						FB_Move.BCGapMove:=TRUE;
						FB_Move();
						HysteresisMoving:=TRUE;		
						n_state:=1;	
					END_IF
				1:
					btn_UserGapMove:=FALSE;
					FB_Move();
					IF NOT FB_Move.BCGapDone THEN			(*还未运动到位置,运动过程中*)
						Led_Run:=TRUE;
						n_state:=1;
					ELSE									
						n_state:=2;							(*转到下一步，运动到最终位置*)
						FB_Move.BCGapMove:=FALSE;
						//Led_Run:=FALSE;
					END_IF
				2:
					FB_Move.BCGapReset:=FALSE;
					FB_Move.Mode:=5;						//1.gap;2.single;3.taper;4.debug;5.BCGap&UserMode
					FB_Move.CoupleState:=st_Couple;			
					FB_Move.PowerState:=st_Power;			
					FB_Move.BCGapMove:=TRUE;
					//直接走到目标位置，已经走到位置的，可以继续下命令，只不过它不在走了而已
					FB_Move.BCLeftTopPosition:=LeftTopLinPositionNewTemp;	
					FB_Move.BCRightTopPosition:=RightTopLinPositionNewTemp;
					FB_Move.BCLeftBottomPosition:=LeftBottomLinPositionNewTemp;
					FB_Move.BCRightBottomPosition:=RightBottomLinPositionNewTemp;
					//
					//目标速度赋值
					IF NormalGapMode THEN
						FB_Move.BCLeftTopVelocity:=UserGapVelocityNew/2;
						FB_Move.BCRightTopVelocity:=UserGapVelocityNew/2;
						FB_Move.BCLeftBottomVelocity:=UserGapVelocityNew/2;
						FB_Move.BCRightBottomVelocity:=UserGapVelocityNew/2;
					ELSIF IDTaperMode THEN
						FB_Move.BCLeftTopVelocity:=UserTaperVelocityNew/2;
						FB_Move.BCRightTopVelocity:=UserTaperVelocityNew/2;
						FB_Move.BCLeftBottomVelocity:=UserTaperVelocityNew/2;
						FB_Move.BCRightBottomVelocity:=UserTaperVelocityNew/2;
					ELSIF BLTaperMode THEN
						FB_Move.BCLeftTopVelocity:=BLUserTaperVelocityNew*IDTaperAndBLTaperScale/4;
						FB_Move.BCRightTopVelocity:=BLUserTaperVelocityNew*IDTaperAndBLTaperScale/4;
						FB_Move.BCLeftBottomVelocity:=BLUserTaperVelocityNew*IDTaperAndBLTaperScale/4;
						FB_Move.BCRightBottomVelocity:=BLUserTaperVelocityNew*IDTaperAndBLTaperScale/4;
					ELSE
						FB_Move.BCLeftTopVelocity:=0;
						FB_Move.BCRightTopVelocity:=0;
						FB_Move.BCLeftBottomVelocity:=0;
						FB_Move.BCRightBottomVelocity:=0;
					END_IF
					FB_Move();							
					n_state:=3;
				3:
					FB_Move();
					IF NOT FB_Move.BCGapDone THEN			(*还未运动到位置,运动过程中*)
						Led_Run:=TRUE;
						n_state:=3;
					ELSE									
						n_state:=88;							(*运动到了最终位置*)
					END_IF
					(*
					IF NOT Unreach_LS_Bottom THEN
						n_state:=88;							(*在运动过程中如果碰到下限位，则也转到下一步，运动到最终位置*)
						FB_Move.BCGapMove_2:=FALSE;
					END_IF
					*)
				88:
					btn_UserGapMove:=FALSE;					
					Led_Run:=FALSE;
					n_state:=0;
					HysteresisMoving:=FALSE;
			END_CASE
		END_IF
	//
	//FB_Move.BCLeftTopPosition等四轴位置监控
	//
END_IF

IF btn_UserGapStop OR btn_Reset THEN
	FB_Move.BCGapReset:=TRUE;
	FB_Move();	
	btn_UserGapMove:=FALSE;	
	m_state:=0;	
	n_state:=0;	
	HysteresisMoving:=FALSE;
	CASE s_state OF
			0:
				FB_Stop.Mode:=5;	
				FB_Stop.CoupleState:=st_Couple;	
				FB_Stop.PowerState:=st_Power;
				FB_Stop.BCGapStop:=TRUE;
				FB_Stop();	
				s_state:=1;
			1:
				FB_Stop();
				IF NOT FB_Stop.BCGapDone THEN
					s_state:=1;
				ELSE
					s_state:=88;
				END_IF
			88:
				btn_UserGapStop:=FALSE;	
				FB_Move.BCGapReset:=FALSE;
				btn_reset:=FALSE;
				s_state:=0;
		END_CASE
END_IF

(*触发限位开关后，相当于点击了Stop按钮*)
FTrig_ReachLS(CLK:=Unreach_LS_Far AND Unreach_LS_Near);
IF FTrig_ReachLS.Q THEN
	btn_UserGapStop:=TRUE;
END_IF
END_ACTION

ACTION A_SpectroscopyScanningMotion:
(*输入保护*)
IF SS_Move AND SSMotionMode AND NOT RegularMotionMode THEN
	IF NOT inRange_SS_StepSize THEN
		SS_Stop:=TRUE;
		SS_Move:=FALSE;
		Error:=TRUE;
		ErrorId:=805;
		ErrorDescription:='target StepSize out of range,please check';
		RETURN;
	ELSE
		//SS_Stop:=FALSE;
		Error:=FALSE;
		ErrorId:=0;
		ErrorDescription:='';	
	END_IF
	//
	IF NOT inRange_SS_StepNumber THEN
		SS_Stop:=TRUE;
		SS_Move:=FALSE;
		Error:=TRUE;
		ErrorId:=806;
		ErrorDescription:='target StepNumber out of range,please check';
		RETURN;
	ELSE
		//SS_Stop:=FALSE;
		Error:=FALSE;
		ErrorId:=0;
		ErrorDescription:='';	
	END_IF
	IF NOT inRange_SS_StepVelocity THEN
		SS_Stop:=TRUE;
		SS_Move:=FALSE;
		Error:=TRUE;
		ErrorId:=807;
		ErrorDescription:='target StepVelocity out of range,please check';
		RETURN;
	ELSE
		//SS_Stop:=FALSE;
		Error:=FALSE;
		ErrorId:=0;
		ErrorDescription:='';	
	END_IF
	IF NOT inRange_StepEachTime_ms THEN
		SS_Stop:=TRUE;
		SS_Move:=FALSE;
		Error:=TRUE;
		ErrorId:=808;
		ErrorDescription:='target StepEachTime_ms out of range,please check';
		RETURN;
	ELSE
		//SS_Stop:=FALSE;
		Error:=FALSE;
		ErrorId:=0;
		ErrorDescription:='';	
	END_IF
END_IF
(*单步时长转换*)
StepEachTime:=INT_TO_TIME(StepEachTime_ms);
SS_TON(PT:=StepEachTime);
(*上升沿触发，初始SS位置=当前磁间隙*)
RTRG_SS_StartPositionDisplay(CLK:=SS_Move);
IF RTRG_SS_StartPositionDisplay.Q THEN
	SS_StartPositionDisplay:=UserGapPositionDisplay;
	SS_InitStartPositionDone:=TRUE;
END_IF
(*SS主程序*)
IF InitPowerDone AND InitCompensationDatasDone AND SS_Move AND SS_InitStartPositionDone THEN
	IF NOT st_Power THEN
		ErrorID:=1501;
		Error:=TRUE;
		ErrorDescription:='Plz PowerOn Frist';
		LED_Error:=TRUE;
		//btn_UserGapMove:=FALSE;
		RETURN;
	ELSE
		ErrorID:=0;
		Error:=FALSE;
		ErrorDescription:='';
		LED_Error:=FALSE;
		//btn_UserGapMove:=TRUE;
	END_IF	
CASE SS_MoveState OF
		0:
				//UserGapPositionNew:=UserGapPositionDisplay+SS_StepSize;
				UserGapPositionNew:=SS_StartPositionDisplay+SS_StepSize*(SS_currentStep+1);
				A_InitCompensationData();
				FB_Move.Mode:=5;						//1.gap;2.single;3.taper;4.debug;5.BCGap&UserMode
				FB_Move.CoupleState:=st_Couple;			
				FB_Move.PowerState:=st_Power;							
				FB_Move.BCLeftTopPosition:=LeftTopLinPositionNew;
				FB_Move.BCLeftTopVelocity:=SS_StepVelocity/2;
				FB_Move.BCRightTopPosition:=RightTopLinPositionNew;
				FB_Move.BCRightTopVelocity:=SS_StepVelocity/2;
				FB_Move.BCLeftBottomPosition:=LeftBottomLinPositionNew;
				FB_Move.BCLeftBottomVelocity:=SS_StepVelocity/2;
				FB_Move.BCRightBottomPosition:=RightBottomLinPositionNew;
				FB_Move.BCRightBottomVelocity:=SS_StepVelocity/2;		
				FB_Move.BCGapMove:=TRUE;
				FB_Move();
				SS_MoveState:=1;
		1:
				SS_TON.IN:=TRUE;
				FB_Move();
				IF FB_Move.GapMoving AND NOT SS_TimeCountBegin THEN
					SS_StepSystemTime_Begin[SS_currentStep]:=F_GetSysTime();
					SS_TimeCountBegin:=TRUE;
				END_IF
				IF NOT FB_Move.BCGapDone THEN			
					Led_Run:=TRUE;
					SS_MoveState:=1;
				ELSE									
					SS_MoveState:=66;
					SS_StepSystemTime_End[SS_currentStep]:=F_GetSysTime();
					SS_StepCountTime[SS_currentStep]:=SS_StepSystemTime_End[SS_currentStep]-SS_StepSystemTime_Begin[SS_currentStep];
					SS_TimeCountBegin:=FALSE;
				END_IF
		66:
				SS_currentStep:=SS_currentStep+1;			
				Led_Run:=FALSE;
				IF SS_currentStep=SS_StepNumber THEN								
					SS_MoveState:=88;
				END_IF
				IF SS_currentStep<SS_StepNumber THEN
					SS_MoveState:=77;
				END_IF
		77://等待单步时长够
				IF SS_TON.Q THEN
					SS_TON.IN:=FALSE;
					SS_MoveState:=0;
				END_IF
		88:
				SS_TON.IN:=FALSE;
				SS_Move:=FALSE;	
				Led_Run:=FALSE;
				SS_MoveState:=0;
				SS_currentStep:=0;
				SS_InitStartPositionDone:=FALSE;
				//SS_StepSystemTime[SS_StepNumber]:=F_GetSysTime();
	END_CASE
END_IF
(*获取每一步耗时*)
//FOR	m:= 0 TO SS_StepNumber DO
//	SS_StepCountTime[m]:=(SS_StepSystemTime_End[m]-SS_StepSystemTime_Begin[m]);
//END_FOR

(*STOP*)
IF SS_Stop OR btn_reset THEN
	FB_Move.BCGapReset:=TRUE;
	FB_Move();	
	SS_Move:=FALSE;	
	SS_MoveState:=0;	
	CASE SS_StopState OF
			0:
				FB_Stop.Mode:=5;						
				FB_Stop.CoupleState:=st_Couple;		
				FB_Stop.PowerState:=st_Power;			
				FB_Stop.BCGapStop:=TRUE;			
				FB_Stop();						
				SS_StopState:=1;
			1:
				FB_Stop();
				IF NOT FB_Stop.BCGapDone THEN		
					SS_StopState:=1;
				ELSE							
					SS_StopState:=88;
				END_IF
			88:
				SS_Stop:=FALSE;					
				FB_Move.BCGapReset:=FALSE;		
				SS_StopState:=0;
				btn_reset:=FALSE;
				//SS_Stop2:=FALSE;
		END_CASE
END_IF

(*触发限位开关后，相当于点击了Stop按钮*)
FTrig_ReachLS(CLK:=Unreach_LS_Far AND Unreach_LS_Near);
IF FTrig_ReachLS.Q THEN
	SS_Stop:=TRUE;
END_IF
END_ACTION

ACTION A_TaperMotionProtection:
(*如果该ID没有taper需求，则TaperFunctionSolidOn=FALSE，则判定taperOrNot和BLTaperOrNot都为FALSE*)
IF NOT TaperFunctionSolidOn THEN
	TaperOrNot:=FALSE;
	BLTaperOrNot:=FALSE;
END_IF
(*若GAP将有变化，首先检测TAPER是否超出阈值，若超出，则报错，提示必须先将TAPER回归到0，才可以改变GAP*)
IF NormalGapMode OR IDTaperMode THEN 
	IF NOT (Global_ChainProtection_MPS_Triggered OR Global_ChainProtection_EPS_Triggered) THEN//在触发联锁保护后，taper保护关闭
		IF ABS(UserGapPositionNew-UserGapPositionDisplay)>Threshold_GapChangeFlag AND btn_UserGapMove THEN
			IF UserTaperPositionDisplay>Threshold_TaperChangeFlag THEN
				btn_UserGapStop:=TRUE;
				btn_UserGapMove:=FALSE;
				Error:=TRUE;
				ErrorId:=809;
				ErrorDescription:='Please Move Taper to zero first before move gap';
				RETURN;
			END_IF
		END_IF
	END_IF
END_IF
IF BLTaperMode THEN
		IF NOT (Global_ChainProtection_MPS_Triggered OR Global_ChainProtection_EPS_Triggered) THEN//在触发联锁保护后，taper保护关闭
		IF ABS(UserGapPositionNew-UserGapPositionDisplay)>Threshold_GapChangeFlag AND btn_UserGapMove THEN
			IF BLUserTaperPositionDisplay>Threshold_TaperChangeFlag THEN
				btn_UserGapStop:=TRUE;
				btn_UserGapMove:=FALSE;
				Error:=TRUE;
				ErrorId:=810;
				ErrorDescription:='Please Move Taper to zero first before move gap';
				RETURN;
			END_IF
		END_IF
	END_IF
END_IF
(*若GAP将有变化,检测taper功能开关有没有关，要是没有关，提示先关闭*)
IF NOT (Global_ChainProtection_MPS_Triggered OR Global_ChainProtection_EPS_Triggered) THEN//在触发联锁保护后，taper保护关闭
	IF ABS(UserGapPositionNew-UserGapPositionDisplay)>Threshold_GapChangeFlag AND btn_UserGapMove THEN
		IF TaperOrNot OR BLTaperOrNot THEN
			btn_UserGapStop:=TRUE;
			btn_UserGapMove:=FALSE;
			Error:=TRUE;
			ErrorId:=811;
			ErrorDescription:='Please turn off taper function before move gap';
			RETURN;
		END_IF
	END_IF
END_IF
(*Taper和gap连锁限制性保护。比如11mm时候如果taper，入口端gap变小，会有压真空盒的问题。设置保护；在大间隙同样保护*)
IF IDTaperMode THEN
	IF NOT (Global_ChainProtection_MPS_Triggered OR Global_ChainProtection_EPS_Triggered)  THEN//在触发联锁保护后，taper保护关闭
		IF UserGapPositionNew-TaperAndGapSafetyfactor*TaperAndGapSafetyScale*UserTaperPositionNew<(min_UserGapPositionNew+TaperAndGapSafetyMinGapMargin)
			OR UserGapPositionNew+TaperAndGapSafetyfactor*TaperAndGapSafetyScale*UserTaperPositionNew>(max_UserGapPositionNew-TaperAndGapSafetyMinGapMargin) THEN
				 IF btn_UserGapMove THEN
					btn_UserGapStop:=TRUE;
					btn_UserGapMove:=FALSE;
					Error:=TRUE;
					ErrorId:=812;
					ErrorDescription:='Target taper is too big at current Gap';
					RETURN;
				END_IF
		END_IF
	END_IF
END_IF
IF BLTaperMode THEN
	IF NOT (Global_ChainProtection_MPS_Triggered OR Global_ChainProtection_EPS_Triggered)  THEN//在触发联锁保护后，taper保护关闭
		IF UserGapPositionNew-BLUserTaperPositionNew/2<(min_UserGapPositionNew+TaperAndGapSafetyMinGapMargin)
			OR UserGapPositionNew+BLUserTaperPositionNew/2>(max_UserGapPositionNew-TaperAndGapSafetyMinGapMargin) THEN
				 IF btn_UserGapMove THEN
					btn_UserGapStop:=TRUE;
					btn_UserGapMove:=FALSE;
					Error:=TRUE;
					ErrorId:=813;
					ErrorDescription:='Target taper is too big at current Gap';
					RETURN;
				END_IF
		END_IF
	END_IF
END_IF
(*Taper和gap连锁限制性保护。大间隙taper过大，有触碰真空盒问题，保护*)
END_ACTION

ACTION A_TaperParametersInit:
// 先做模式判断
NormalGapMode := NOT TaperOrNot AND NOT BLTaperOrNot;
IDTaperMode := TaperOrNot AND NOT BLTaperOrNot;
BLTaperMode := NOT TaperOrNot AND BLTaperOrNot;
//TaperOrNot和BLTaperOrNot互斥，只能选择其中一个
trig_TaperOrNot(CLK := TaperOrNot);
trig_BLTaperOrNot(CLK := BLTaperOrNot);
IF trig_TaperOrNot.Q THEN
    BLTaperOrNot := FALSE;
ELSIF trig_BLTaperOrNot.Q THEN
    TaperOrNot := FALSE;
END_IF;

//插入件taper/线站taper
IDTaperAndBLTaperScale:=L_Center2Motor/L_HalfGirder;
//插入件taper模式下，入口被动减小的距离，也即a
TaperAndGapSafetyScale:=DINT_TO_LREAL(LREAL_TO_DINT(((L_HalfGirder-L_Center2Motor)/(2*L_Center2Motor))*100000))/100000;

//线站模式下，最大taper由参数表决定，ID模式的最大tape由scale计算得到
max_UserTaperPositionNew:=DINT_TO_LREAL(LREAL_TO_DINT((max_BLUserTaperPositionNew*IDTaperAndBLTaperScale)*100000))/100000;
max_UserTaperVelocityNew:=DINT_TO_LREAL(LREAL_TO_DINT((max_BLUserTaperVelocityNew)*100000))/100000;
//最小taper固定位0
min_UserTaperPositionNew:=0;
min_UserTaperVelocityNew:=0;
END_ACTION

END_PROGRAM

// ---- POUs/MAIN.TcPOU
PROGRAM MAIN
VAR
	pbGapMode: BOOL:=FALSE;
	pbTaperMode: BOOL:=FALSE;
	pbSingleCarrierMode: BOOL:=FALSE;
	pbDebugMode:BOOL:=FALSE;
	pbBCGapMode:BOOL:=FALSE;
	fb_led_Show: FB_LedShow;
	CPMU_PLC_Reset: PLC_Reset;
	d_state: DINT;
	CPMU_PLC_Start: PLC_Start;
	powerStatus:BOOL;

(*TwinSAFE*)
	Safe_run AT%Q*:BOOL;
	Err_Ack AT %Q*:BOOL;
	Estop_RunAndRestart AT %Q*:BOOL;
	AX5805_Error_Ack AT %Q*:BOOL;
	Led_Run  AT %Q*:BOOL;
	Led_Error  AT %Q*:BOOL;

	FB_ERROR AT%I*:BOOL;
	COM_ERROR AT%I*:BOOL;
	//OUT_ERROR AT%I*:BOOL;
	Estop_Out AT%I*:BOOL;

	SafeStatus:INT;
	SafePLCRunOK: BOOL;
	fb_ton: TON;
	fb_ton2: TON;
	fb_ton3: TON;
	fb_ton1: TON;
	fb_ton0: TON;
(*IO*)
	el1808_D1  AT%I* :ARRAY[1..8] OF BOOL;
	el1008 AT%I*:BOOL;
	EStopTrig:BOOL;
(*setAxisPosition*)
	SetAxisPosState: INT;
	FB_Set_AxisPosition:FB_SetAxisPosition;
	fb_ton4: TON;
	fb_ton5: TON;
	fb_ton6: TON;
	SerAxisPositionDone: BOOL;

	i: INT;
	j: INT;

(****RS232***)
	//fbEL6001	: FB_SerialCom;
	moveDoneLeftTop: BOOL;
	moveDoneRightTop: BOOL;
	moveDoneLeftBottom: BOOL;
	moveDoneRightBottom: BOOL;
	moveDoneAllAxis: BOOL;
(**)
	btn_setAxisPosition: BOOL;
	ValueSet_LeftTop:LREAL;
	ValueSet_RightTop:LREAL;
	ValueSet_LeftBottom:LREAL;
	ValueSet_RightBottom:LREAL;
(**)
	RestartTC: TC_Restart;
	
(*recipe*)
	RecipeINT:INT;
	RecipeBOOL:BOOL;
	RecipeManCommands: RecipeManCommands;
	SaveParameter : BOOL;  //保存文件
	LoadParameter : BOOL;  //读取文件
	Save_R_TRIG   : R_TRIG;
	Read_R_TRIG   : R_TRIG;
	loadparameterStatus: INT;
	RecipeBOOL2:BOOL;
	ReturnDwordLoad: DWORD;
	InsertionDeviceName:STRING;
(*UserMode*)
	pbUserMode: BOOL:=TRUE;
	EL1904 AT%I* :ARRAY[1..24] OF BOOL;
	setAxisPositionEnable: BOOL;
	state_loadParameters: INT;
	state_setLEPosBias: INT;
	//
	PositionBiasSet:BOOL;
	MC_SetLEPosBias_LeftTop:MC_WriteParameter;
	MC_SetLEPosBias_RightTop:MC_WriteParameter;
	MC_SetLEPosBias_LeftBottom:MC_WriteParameter;
	MC_SetLEPosBias_RightBottom:MC_WriteParameter;
	PositionBias_LeftTopLin: LREAL:=10.1;
	PositionBias_RightTopLin: LREAL:=10.2;
	PositionBias_LeftBottomLin: LREAL:=10.3;
	PositionBias_RightBottomLin: LREAL:=10.4;
	PositionBias_LeftTop: LREAL:=10.1;
	PositionBias_RightTop: LREAL:=10.2;
	PositionBias_LeftBottom: LREAL:=10.3;
	PositionBias_RightBottom: LREAL:=10.4;

	LoadLEPB_R_TRIG: R_TRIG;
	PositionBiasTON: TON;
	
	//
	OPC_TEST_Bi:BOOL:=TRUE; (*~ (OPC:1:available for OPC Clients) *)
	OPC_TEST_Bi2:BOOL;(*~ (OPC:1:available for OPC Clients) *)
	//
	HasTemperatureSensorOrNot:BOOL;//Only IVU or CPMU
	(*Sensor Reading*)
	TempSensorHardware:DINT:=1;//1:profibus;2:EL3202
	EL3202_Reading AT %I*:ARRAY[0..7] OF INT;	
	EL3202_hReading AT %I*:ARRAY[0..7] OF INT;
	Sensor_Reading_1 AT %I*:ARRAY[0..3] OF BYTE;
	Sensor_Reading_2 AT %I*:ARRAY[0..3] OF BYTE;
	Sensor_Reading_3 AT %I*:ARRAY[0..3] OF BYTE;
	Sensor_Reading_4 AT %I*:ARRAY[0..3] OF BYTE;
	Sensor_Reading_5 AT %I*:ARRAY[0..3] OF BYTE;
	Sensor_Reading_6 AT %I*:ARRAY[0..3] OF BYTE;
	Sensor_Reading_7 AT %I*:ARRAY[0..3] OF BYTE;
	Sensor_Reading_8 AT %I*:ARRAY[0..3] OF BYTE;
	Sensor_Reading_DpState AT %I*:USINT;
	Sensor_Reading_ExtDiagFlag AT %I*:BOOL;
	TemperatureSensors_1:LREAL;
	TemperatureSensors_2:LREAL;
	TemperatureSensors_3:LREAL;
	TemperatureSensors_4:LREAL;
	TemperatureSensors_5:LREAL;
	TemperatureSensors_6:LREAL;
	TemperatureSensors_7:LREAL;
	TemperatureSensors_8:LREAL;
	dut_sensor_datas_1:DUT_SENSOR_DATAS_1;
	dut_sensor_datas_2:DUT_SENSOR_DATAS_2;
	dut_sensor_datas_3:DUT_SENSOR_DATAS_3;
	dut_sensor_datas_4:DUT_SENSOR_DATAS_4;
	dut_sensor_datas_5:DUT_SENSOR_DATAS_5;
	dut_sensor_datas_6:DUT_SENSOR_DATAS_6;
	dut_sensor_datas_7:DUT_SENSOR_DATAS_7;
	dut_sensor_datas_8:DUT_SENSOR_DATAS_8;
	//
	temperature_gradient_2_To_1:LREAL;
	temperature_gradient_3_To_2:LREAL;
	temperature_gradient_5_To_4:LREAL;
	temperature_gradient_6_To_5:LREAL;
	temperature_gradient_max:LREAL;
	//
	temperature_average:LREAL;
	A_SetLinearEncoderPositionBias_Enable: BOOL;
	
	//
	//(*Sensor Reading high temperature*)
	//
	Sensor_Reading_h1 AT %I*:ARRAY[0..3] OF BYTE;
	Sensor_Reading_h2 AT %I*:ARRAY[0..3] OF BYTE;
	Sensor_Reading_h3 AT %I*:ARRAY[0..3] OF BYTE;
	Sensor_Reading_h4 AT %I*:ARRAY[0..3] OF BYTE;
	Sensor_Reading_h5 AT %I*:ARRAY[0..3] OF BYTE;
	Sensor_Reading_h6 AT %I*:ARRAY[0..3] OF BYTE;
	Sensor_Reading_h7 AT %I*:ARRAY[0..3] OF BYTE;
	Sensor_Reading_h8 AT %I*:ARRAY[0..3] OF BYTE;
	Sensor_Reading_DpStateh AT %I*:USINT;
	Sensor_Reading_ExtDiagFlagh AT %I*:BOOL;
	TemperatureSensors_h1:LREAL;
	TemperatureSensors_h2:LREAL;
	TemperatureSensors_h3:LREAL;
	TemperatureSensors_h4:LREAL;
	TemperatureSensors_h5:LREAL;
	TemperatureSensors_h6:LREAL;
	TemperatureSensors_h7:LREAL;
	TemperatureSensors_h8:LREAL;
	dut_sensor_datas_h1:DUT_SENSOR_DATAS_h1;
	dut_sensor_datas_h2:DUT_SENSOR_DATAS_h2;
	dut_sensor_datas_h3:DUT_SENSOR_DATAS_h3;
	dut_sensor_datas_h4:DUT_SENSOR_DATAS_h4;
	dut_sensor_datas_h5:DUT_SENSOR_DATAS_h5;
	dut_sensor_datas_h6:DUT_SENSOR_DATAS_h6;
	dut_sensor_datas_h7:DUT_SENSOR_DATAS_h7;
	dut_sensor_datas_h8:DUT_SENSOR_DATAS_h8;
	//
	temperature_gradient_h2_To_h1:LREAL;
	temperature_gradient_h3_To_h2:LREAL;
	temperature_gradient_h5_To_h4:LREAL;
	temperature_gradient_h6_To_h5:LREAL;
	temperature_gradient_maxh:LREAL;
	//
	temperature_averageh:LREAL;
		//
	temperatureStatus:INT;//0：有传感器度数错误；1:常温；2:低温；3:常温和低温中间态
	CryogenicTemperatureThreshold:LREAL:=82;//82K以下归划分为低温
	RoomTemperatureThreshold:LREAL:=293;//293K以上划分为常温.20摄氏度
	InCryogenicOrNot:BOOL;
	//CPMU cryogenix ON/FF
	CryogenicCompensationOn:BOOL;
	CryogenicCompensationConditionsReady:BOOL;
	CryogenicCompensation_LeftTop:LREAL;
	CryogenicCompensation_RightTop:LREAL;
	CryogenicCompensation_LeftBottom:LREAL;
	CryogenicCompensation_RightBottom:LREAL;
	CryogenicCompensationDone: BOOL;
	
	(**)
	bDriveDiagMessageAndNumber  : BOOL;
	m_GetDriveStatusState:INT;
	GetDriveStatusStateDone:BOOL;
	GetDriveStatusStateError:BOOL;
	GetDriveStatusTON: TON;
	//	
	fb_SoEReadDiagMessage_LeftTop: FB_SoEReadDiagMessage;
	fb_SoEReadDiagMessage_RightTop: FB_SoEReadDiagMessage;
	fb_SoEReadDiagMessage_LeftBottom: FB_SoEReadDiagMessage;
	fb_SoEReadDiagMessage_RightBottom: FB_SoEReadDiagMessage;
	DriveDiagMessage_LeftTop:STRING;
	DriveDiagMessage_RightTop:STRING;
	DriveDiagMessage_LeftBottom:STRING;
	DriveDiagMessage_RightBottom:STRING;
	//
	FB_SoEReadDiagNumber_LeftTop: FB_SoEReadDiagNumber;
	FB_SoEReadDiagNumber_RightTop: FB_SoEReadDiagNumber;
	FB_SoEReadDiagNumber_LeftBottom: FB_SoEReadDiagNumber;
	FB_SoEReadDiagNumber_RightBottom: FB_SoEReadDiagNumber;
	DriveDiagNumber_LeftTop:UDINT;
	DriveDiagNumber_RightTop:UDINT;
	DriveDiagNumber_LeftBottom:UDINT;
	DriveDiagNumber_RightBottom:UDINT;
	bReloadDriveDiagMessageAndNumber: BOOL;
	
	(*load IOC*)
	bExe_load_Prog: BOOL;
	NT_StartProcess_Load: NT_StartProcess;
	Exe_load_step: UINT;
	R_TRIG_ExeLoad: R_TRIG;
	Exe_Load_Done:BOOL;
	(*kill IOC*)
	bExe_Kill_Prog: BOOL;
	NT_StartProcess_Kill: NT_StartProcess;
	Exe_kill_step: UINT;
	R_TRIG_Exekill: R_TRIG;
	Exe_Kill_Done:BOOL;
	LoadOpcIocTON:TON;
	
	LeftTop_2:AXIS_REF;
	RightTop_2:AXIS_REF;
	LeftBottom_2:AXIS_REF;
	RightBottom_2:AXIS_REF;
	Pos_LeftTop_2:LREAL;
	Velo_LeftTop_2:LREAL;
	Pos_RightTop_2:LREAL;
	Velo_RightTop_2:LREAL;
	Pos_LeftBottom_2:LREAL;
	Velo_LeftBottom_2:LREAL;
	Pos_RightBottom_2:LREAL;
	Velo_RightBottom_2:LREAL;
	PosDifference_LeftTop2to1:LREAL;
	PosDifference_RightTop2to1:LREAL;
	PosDifference_LeftBottom2to1:LREAL;
	PosDifference_RightBottom2to1:LREAL;
	//
	//more parameters get:gear;feedback2 direction 
	//
	//GetMoreDriveStatus_FunctionON:BOOL:=TRUE;
	GetDriveStatusTON2: TON;
	//GearNumerator,st182
	st_p182_LeftTop:ST_P182;
	FB_SoERead_GearNumerator_LeftTop: FB_SoERead;
	st_p182_RightTop:ST_P182;
	FB_SoERead_GearNumerator_RightTop: FB_SoERead;
	st_p182_LeftBottom:ST_P182;
	FB_SoERead_GearNumerator_LeftBottom: FB_SoERead;
	st_p182_RightBottom:ST_P182;
	FB_SoERead_GearNumerator_RightBottom: FB_SoERead;
	GearNumeratorGet_LeftTop:UDINT;
	GearNumeratorGet_RightTop:UDINT;
	GearNumeratorGet_LeftBottom:UDINT;
	GearNumeratorGet_RightBottom:UDINT;
	GearNumeratorConfigured_LeftTop:UDINT;
	GearNumeratorConfigured_RightTop:UDINT;
	GearNumeratorConfigured_LeftBottom:UDINT;
	GearNumeratorConfigured_RightBottom:UDINT;
	//GearDenominator,st183
	st_p183_LeftTop:ST_P183;
	FB_SoERead_GearDenominator_LeftTop: FB_SoERead;
	st_p183_RightTop:ST_P183;
	FB_SoERead_GearDenominator_RightTop: FB_SoERead;
	st_p183_LeftBottom:ST_P183;
	FB_SoERead_GearDenominator_LeftBottom: FB_SoERead;
	st_p183_RightBottom:ST_P183;
	FB_SoERead_GearDenominator_RightBottom: FB_SoERead;
	GearDenominatorGet_LeftTop:UDINT;
	GearDenominatorGet_RightTop:UDINT;
	GearDenominatorGet_LeftBottom:UDINT;
	GearDenominatorGet_RightBottom:UDINT;
	GearDenominatorConfigured_LeftTop:UDINT;
	GearDenominatorConfigured_RightTop:UDINT;
	GearDenominatorConfigured_LeftBottom:UDINT;
	GearDenominatorConfigured_RightBottom:UDINT;
	//Feedback2direction,st180
	st_p180_LeftTop:ST_P180;
	FB_SoERead_Feedback2direction_LeftTop: FB_SoERead;
	st_p180_RightTop:ST_P180;
	FB_SoERead_Feedback2direction_RightTop: FB_SoERead;
	st_p180_LeftBottom:ST_P180;
	FB_SoERead_Feedback2direction_LeftBottom: FB_SoERead;
	st_p180_RightBottom:ST_P180;
	FB_SoERead_Feedback2direction_RightBottom: FB_SoERead;
	Feedback2directionGet_LeftTop:UINT;
	Feedback2directionGet_RightTop:UINT;
	Feedback2directionGet_LeftBottom:UINT;
	Feedback2directionGet_RightBottom:UINT;
	Feedback2directionConfigured_LeftTop:UINT;
	Feedback2directionConfigured_RightTop:UINT;
	Feedback2directionConfigured_LeftBottom:UINT;
	Feedback2directionConfigured_RightBottom:UINT;
	//
	//RestartDrivers
		(*重启驱动器*)
	btn_RestartDriversAll:BOOL;
	btn_RestartDriver1:BOOL;
	btn_RestartDriver2:BOOL;
	btn_RestartDriver3:BOOL;
	btn_RestartDriver4:BOOL;
	btn_RestartDriver5:BOOL;
	btn_RestartDriver6:BOOL;
	btn_RestartDriver7:BOOL;
	btn_RestartDriver8:BOOL;
	Relay_EL2624 AT %Q*:ARRAY[0..7]OF  BOOL;
	RestartDriver_RTRIG:R_TRIG;
	RestartDriver_TON:TON;
	RestartDriver_Triggered:BOOL;
	RestartDriver_State:DINT;
	RestartDriver_Done:BOOL;

	//
	//	LEHeartBeatMonitorFunction
	//
	LEHeartBeatMonitorFunctionOn: BOOL;
	LEHeartBeatFirstScan:BOOL;
	LEHeartBeatDeadZone : LREAL := 0; 
	LEHeartBeatAlarmTime : TIME := T#0.1S;
	
    //Pos_LeftTopLin_Last : LREAL; 
	Velo_LeftTopLin_Last : LREAL; 
	Pos_LeftTopMotor_Initial : LREAL; 
    StableTimer_LeftTopLin : TON; 
    StableTime_LeftTopLin : TIME; 
    DeltaVelo_LeftTopLin : LREAL; 
	IsInitialPositionSet_LeftTop: BOOL;
	MotorPosChange_LeftTop: LREAL;
	Threshold_LeftTopMotorPos:LREAL:=0.1;
	Threshold_LeftTopMotorVelo:LREAL:=0.2;
	Alarm_LeftTopLin:BOOL;
	Alarm_LeftTopMotorPos:BOOL;
	Alarm_LeftTopMotorVelo:BOOL;
	
	
	//Pos_RightTopLin_Last : LREAL; 
	Velo_RightTopLin_Last : LREAL; 
	Pos_RightTopMotor_Initial : LREAL; 
    StableTimer_RightTopLin : TON; 
    StableTime_RightTopLin : TIME; 
    DeltaVelo_RightTopLin : LREAL; 
	IsInitialPositionSet_RightTop: BOOL;
	MotorPosChange_RightTop: LREAL; 
	Threshold_RightTopMotorPos:LREAL:=0.1;
	Threshold_RightTopMotorVelo:LREAL:=0.2;
	Alarm_RightTopLin:BOOL;
	Alarm_RightTopMotorPos:BOOL;
	Alarm_RightTopMotorVelo:BOOL;
	
		
    //Pos_LeftBottomLin_Last : LREAL; 
	Velo_LeftBottomLin_Last : LREAL; 
	Pos_LeftBottomMotor_Initial : LREAL; 
    StableTimer_LeftBottomLin : TON; 
    StableTime_LeftBottomLin : TIME; 
    DeltaVelo_LeftBottomLin : LREAL; 
	IsInitialPositionSet_LeftBottom: BOOL;
	MotorPosChange_LeftBottom: LREAL; 
	Threshold_LeftBottomMotorPos:LREAL:=0.1;
	Threshold_LeftBottomMotorVelo:LREAL:=0.2;
	Alarm_LeftBottomLin:BOOL;
	Alarm_LeftBottomMotorPos:BOOL;
	Alarm_LeftBottomMotorVelo:BOOL;
	
	//Pos_RightBottomLin_Last : LREAL; 
	Velo_RightBottomLin_Last : LREAL; 
	Pos_RightBottomMotor_Initial : LREAL; 
    StableTimer_RightBottomLin : TON; 
    StableTime_RightBottomLin : TIME; 
    DeltaVelo_RightBottomLin : LREAL; 
	IsInitialPositionSet_RightBottom: BOOL;
	MotorPosChange_RightBottom: LREAL; 
	Threshold_RightBottomMotorPos:LREAL:=0.1;
	Threshold_RightBottomMotorVelo:LREAL:=0.2;
	Alarm_RightBottomLin:BOOL;
	Alarm_RightBottomMotorPos:BOOL;
	Alarm_RightBottomMotorVelo:BOOL;
	//
	fbMC_ReadParameter_ScaleFactor_LeftTopLIn: MC_ReadParameter;
	fbMC_ReadParameter_ScaleFactor_RightTopLIn: MC_ReadParameter;
	fbMC_ReadParameter_ScaleFactor_LeftBottomLIn: MC_ReadParameter;
	fbMC_ReadParameter_ScaleFactor_RightBottomLIn: MC_ReadParameter;
	ScaleFactor_LeftTopLin: LREAL;
	ScaleFactor_RightTopLin: LREAL;
	ScaleFactor_LeftBottomLin: LREAL;
	ScaleFactor_RightBottomLin: LREAL;
	//
	Velo_LeftTopMotor_DINT AT %I*: DINT;
	Pos_LeftTopMotor_DINT AT %I*: DINT;
	Velo_RightTopMotor_DINT AT %I*: DINT;
	Pos_RightTopMotor_DINT AT %I*: DINT;
	Velo_LeftBottomMotor_DINT AT %I*: DINT;
	Pos_LeftBottomMotor_DINT AT %I*: DINT;
	Velo_RightBottomMotor_DINT AT %I*: DINT;
	Pos_RightBottomMotor_DINT AT %I*: DINT;
	
	(*setAxisPosition*)
	SetMotorAxisPosState: INT;
	FB_Set_MotorAxisPosition:FB_SetMotorAxisPosition;
	fb_ton4_2: TON;
	fb_ton5_2: TON;
	fb_ton6_2: TON;
	SetMotorAxisPositionDone: BOOL;
	
	btn_SetMotorAxisPosition: BOOL;
	MonitorMotorAndLEFunctionOn:BOOL:=TRUE;
	
	{attribute:'TcAnalytics'}
	X:REAL;
	AutoLoadOpcIOC: BOOL:=TRUE;
	(*GetMotorTempture*)
	MotorTemperature AT %I*:ARRAY[0..3] OF UINT;
	MotorTemperature_LeftTop:LREAL;
	MotorTemperature_RightTop:LREAL;
	MotorTemperature_LeftBottom:LREAL;
	MotorTemperature_RightBottom:LREAL;
	
END_VAR

(*MaintenanceMode*)
IF MaintenanceMode THEN
	MaintenanceModeLed:=TRUE;
	RETURN;
ELSE
	MaintenanceModeLed:=FALSE;	
END_IF
(*加载Ricipe参数*)
A_InitRecipeParameters();
IF NOT loadParametersDone THEN
	RETURN;
END_IF
(*Restart TwinCAT*)
IF Global_Variables.m_restartTC THEN
(*首先关闭opcIocShell.exe*)	
	bExe_Kill_Prog:=TRUE;
	A_KillOpcIocShellExe();
(*重启TC*)
	IF Exe_Kill_Done THEN
		RestartTC.RESTART:=TRUE;
		A_RestartTC();
	END_IF
END_IF
//只重启TC，不kill IOC
//IF Global_Variables.m_simpleRestartTC THEN
//	RestartTC.RESTART:=TRUE;
//	A_RestartTC();
//END_IF
(*******InitAxisParameters*******)
A_InitAxisParameters();
(*******CheckLimitSwitch*******)
A_CheckLimitSwitch();
(*Check Kill Switch*)
A_CheckKillSwitch();
(*******PosDiff¼à¿Ø*******)
A_PosDiffDetectiion();
(*******³õÊ¼»¯SafePlc*******)
IF NOT simulation THEN
A_SafePlcStartInit();
END_IF
(************SetAxisPosition*********************)
IF  NOT USELinearEncoder AND setAxisPositionEnable AND btn_setAxisPosition THEN
	//IF NOT SerAxisPositionDone THEN
		FB_Set_AxisPosition.ValueSet_LeftTop:=ValueSet_LeftTop;
		FB_Set_AxisPosition.ValueSet_RightTop:=ValueSet_RightTop;
		FB_Set_AxisPosition.ValueSet_LeftBottom:=ValueSet_LeftBottom;
		FB_Set_AxisPosition.ValueSet_RightBottom:=ValueSet_RightBottom;
		A_SetAxisPosition();
	//END_IF
END_IF
(*******³Mode Select******)
IF SafePLCRunOK OR Simulation THEN
	IF pbSingleCarrierMode AND NOT pbTaperMode AND NOT pbGapMode AND NOT pbDebugMode AND NOT pbBCGapMode AND NOT pbUserMode THEN
		SingleCarrierMode();
	ELSIF pbTaperMode  AND NOT pbSingleCarrierMode AND NOT pbGapMode  AND NOT pbDebugMode AND NOT pbBCGapMode AND NOT pbUserMode THEN
		TaperMode();
	ELSIF pbGapMode AND  NOT pbSingleCarrierMode AND NOT pbTaperMode  AND NOT pbDebugMode AND NOT pbBCGapMode AND NOT pbUserMode THEN
		GapMode();
	ELSIF pbDebugMode AND NOT pbGapMode AND NOT pbSingleCarrierMode AND NOT pbTaperMode AND NOT pbBCGapMode  AND NOT pbUserMode THEN
		DebugMode();
	ELSIF pbBCGapMode AND NOT pbGapMode AND NOT pbSingleCarrierMode AND NOT pbTaperMode AND NOT pbDebugMode AND NOT pbUserMode THEN
		BCGapMode();
	ELSIF pbUserMode AND NOT pbGapMode AND NOT pbSingleCarrierMode AND NOT pbTaperMode AND NOT pbDebugMode AND NOT pbBCGapMode THEN
		UserMode();
	END_IF
END_IF
(*******Led Show******)
fb_led_Show();
(*******Check Power status******)
FB_Power(Check:=TRUE);
st_Power:=FB_Power.PowerState;
(******Check Couple Status*****)
FB_CheckCoupleStatus(Check:=TRUE);
st_Couple:=FB_CheckCoupleStatus.CoupleState;
(*********RS232*********************)
//BackgroundEL();
(*fbEL6001(TxBuffer:=TxBufferEL, RxBuffer:=RxBufferEL);*)

(*获取温度传感器数据*)
A_GetTemperatureSensorsData();
(*低温补偿监控*)
A_CryogenicCompensationMonitoring();

(*设置position bias*)
IF loadParametersDone AND (DriveStatus=1 OR simulation) THEN 
	A_SetLinearEncoderPositionBias();
END_IF
(*检查硬急停状态，包括安全限位、柜门急停、手持急停*)
A_CheckHardwareEmergencyStopStatus();
(*获取驱动器状态信息*)
IF NOT simulation THEN
	A_GetDriverStatus();
END_IF
(*IDControlReady*)
IF ((DriveStatus<>0 AND SafePLCRunOK) OR simulation) AND NOT Error THEN
//IF (SafePLCRunOK OR simulation) AND NOT Error THEN
	IDControlReady:=TRUE;
ELSE
	IDControlReady:=FALSE;
END_IF

(*IOC Start*)
IF AutoLoadOpcIOC THEN
	bExe_load_Prog:=TRUE;
	A_LoadOpcIocShellExe();
END_IF


(*reset*)

(*检查光栅读数是否在范围内*)
A_CheckLinearEncoder();

(*RestartDrivers*)
A_RestartDrivers();

(*ColiControl Function*)
(*Use in HALF *)
IF CoilControlFunction THEN
	PS1();
	PS2();
	PS3();
END_IF

(*A_LEHeartBeatMonitor*)
IF LEHeartBeatMonitorFunctionOn THEN
	A_LEHeartBeatMonitor();
END_IF
(************SetMotorAxisPosition*********************)
//IDControl 1s after
fb_ton5_2.IN:=IDControlReady;
fb_ton5_2.PT:=T#1S;
fb_ton5_2();
IF fb_ton5_2.Q THEN
	btn_SetMotorAxisPosition:=TRUE;
END_IF
IF  USELinearEncoder AND btn_SetMotorAxisPosition THEN
	IF NOT SetMotorAxisPositionDone THEN
		FB_Set_MotorAxisPosition.ValueSet_LeftTop:=Pos_LeftTopLin;
		FB_Set_MotorAxisPosition.ValueSet_RightTop:=Pos_RightTopLin;
		FB_Set_MotorAxisPosition.ValueSet_LeftBottom:=Pos_LeftBottomLin;
		FB_Set_MotorAxisPosition.ValueSet_RightBottom:=Pos_RightBottomLin;
		A_SetMotorAxisPosition();
	END_IF
END_IF
(*A_MonitorMotorAndLE*)
IF MonitorMotorAndLEFunctionOn AND SetMotorAxisPositionDone THEN
	A_MonitorMotorAndLE();
END_IF
(*A_CheckMaxVelocity*)
A_CheckMaxVelocity();
(**)
A_GetMotorTemperature();

ACTION A_CheckHardwareEmergencyStopStatus:
IF 	NOT KS_LeftTop_Far_Contact1 OR
	NOT KS_LeftTop_Far_Contact2 OR
	NOT KS_RightTop_Far_Contact1 OR
	NOT KS_RightTop_Far_Contact2 OR
	NOT KS_LeftBottom_Far_Contact1 OR
	NOT KS_LeftBottom_Far_Contact2 OR
	NOT KS_RightBottom_Far_Contact1 OR
	NOT KS_RightBottom_Far_Contact2 OR
	
	NOT KS_LeftTop_Near_Contact1 OR
	NOT KS_LeftTop_Near_Contact2 OR
	NOT KS_RightTop_Near_Contact1 OR
	NOT KS_RightTop_Near_Contact2 OR
	NOT KS_LeftBottom_Near_Contact1 OR
	NOT KS_LeftBottom_Near_Contact2 OR
	NOT KS_RightBottom_Near_Contact1 OR
	NOT KS_RightBottom_Near_Contact2 OR
(*E-STOP*)
	NOT KS_CabinetEmergency_contact1 OR
	NOT KS_CabinetEmergency_contact2 OR
	NOT KS_handEmergency1_Contact1 OR
	NOT KS_handEmergency1_Contact2 OR
	NOT KS_handEmergency2_Contact1 OR
	NOT KS_handEmergency2_Contact2 OR
	NOT KS_softEmergency2_Contact THEN
	Hardware_EmergencyStop:=FALSE;
ELSE
	Hardware_EmergencyStop:=TRUE;
END_IF
END_ACTION

ACTION A_CheckKillSwitch:
IF simulation THEN
	KS_LeftTop_Far_Contact1:=TRUE;
	KS_LeftTop_Far_Contact2:=TRUE;
	KS_LeftTop_Near_Contact1:=TRUE;
	KS_LeftTop_Near_Contact2:=TRUE;
	KS_RightTop_Far_Contact1:=TRUE;
	KS_RightTop_Far_Contact2:=TRUE;
	KS_RightTop_Near_Contact1:=TRUE;
	KS_RightTop_Near_Contact2:=TRUE;
	KS_LeftBottom_Far_Contact1:=TRUE;
	KS_LeftBottom_Far_Contact2:=TRUE;
	KS_LeftBottom_Near_Contact1:=TRUE;
	KS_LeftBottom_Near_Contact2:=TRUE;	
	KS_RightBottom_Far_Contact1:=TRUE;
	KS_RightBottom_Far_Contact2:=TRUE;
	KS_RightBottom_Near_Contact1:=TRUE;
	KS_RightBottom_Near_Contact2:=TRUE;		
	(*E-STOP*)
	KS_CabinetEmergency_contact1:=TRUE;
	KS_CabinetEmergency_contact2:=TRUE;	
	KS_handEmergency1_Contact1:=TRUE;
	KS_handEmergency1_Contact2:=TRUE;
	KS_handEmergency2_Contact1:=TRUE;
	KS_handEmergency2_Contact2:=TRUE;
	
	KS_softEmergency2_Contact:=TRUE;

ELSE
	KS_LeftTop_Far_Contact1:=EL1904[1];//c1
	KS_LeftTop_Far_Contact2:=EL1904[2];//c2
	KS_LeftTop_Near_Contact1:=EL1904[3];//c3
	KS_LeftTop_Near_Contact2:=EL1904[4];//c4
	
	KS_RightTop_Far_Contact1:=EL1904[5];
	KS_RightTop_Far_Contact2:=EL1904[6];
	KS_RightTop_Near_Contact1:=EL1904[7];
	KS_RightTop_Near_Contact2:=EL1904[8];
	
	KS_LeftBottom_Far_Contact1:=EL1904[9];
	KS_LeftBottom_Far_Contact2:=EL1904[10];
	KS_LeftBottom_Near_Contact1:=EL1904[11];
	KS_LeftBottom_Near_Contact2:=EL1904[12];
	
	KS_RightBottom_Far_Contact1:=EL1904[13];
	KS_RightBottom_Far_Contact2:=EL1904[14];
	KS_RightBottom_Near_Contact1:=EL1904[15];
	KS_RightBottom_Near_Contact2:=EL1904[16];	
	
	
	(*E-STOP*)
	KS_CabinetEmergency_contact1:=EL1904[17];
	KS_CabinetEmergency_contact2:=EL1904[18];
	
	KS_handEmergency1_Contact1:=EL1904[19];
	KS_handEmergency1_Contact2:=EL1904[20];
	KS_handEmergency2_Contact1:=EL1904[21];
	KS_handEmergency2_Contact2:=EL1904[22];
	
	KS_softEmergency2_Contact:=EL1904[23];
	END_IF
END_ACTION

ACTION A_CheckLimitSwitch:
(*******1.´ÓIO»ñÈ¡ÏÞÎ»×´Ì¬******)
(**)
IF simulation THEN
	(**)
	LS_LeftTop_Far:=TRUE;
	LS_LeftTop_Near:=TRUE;
	LS_RightTop_Far:=TRUE;
	LS_RightTop_Near:=TRUE;
	LS_LeftBottom_Far:=TRUE;
	LS_LeftBottom_Near:=TRUE;
	LS_RightBottom_Far:=TRUE;
	LS_RightBottom_Near:=TRUE;
ELSE
	LS_LeftTop_Far :=el1808_D1[1];
	LS_LeftTop_Near:=el1808_D1[3];
	LS_RightTop_Far:=el1808_D1[2];
	LS_RightTop_Near:=el1808_D1[4];
	LS_LeftBottom_Far:=el1808_D1[7];
	LS_LeftBottom_Near:=el1808_D1[5];
	LS_RightBottom_Far:=el1808_D1[8];
	LS_RightBottom_Near:=el1808_D1[6];
END_IF
(*
	LS_LeftTop_Top:=TRUE;
	LS_LeftTop_Bottom:=TRUE;
	LS_RightTop_Top:=TRUE;
	LS_RightTop_Bottom:=TRUE;
	LS_LeftBottom_Top:=TRUE;
	LS_LeftBottom_Bottom:=TRUE;
	LS_RightBottom_Top:=TRUE;
	LS_RightBottom_Bottom:=TRUE;
*)
(******2.TopÏÞÎ»»òÕßBottomÏÞÎ»ÓÐÒ»¸ö´¥·¢£¬È«¾Ö±äÁ¿¡£¸øMC_POWERÓÃÓÚ·½Ïò¿ØÖÆ£¬ÓÐÒ»¸öÏÞÎ»Îª´¥·¢ÎªFALSE£¬ÔòUnreach_LSÎªFALSE******)
Unreach_LS_Far:=LS_LeftTop_Far AND LS_RightTop_Far AND LS_LeftBottom_Far AND LS_RightBottom_Far;
Unreach_LS_Near:=LS_LeftTop_Near AND LS_RightTop_Near AND LS_LeftBottom_Near AND LS_RightBottom_Near;
(**************************ÏòTopÔË¶¯Ê±£¬´¥ÅöBottomÏÞÎ»¿ª¹Ø£¬»òÕßÏà·´£¬ESTOP**************************************)
(*
IF LeftTopLin.Status.Moving AND Velo_LeftTopLin>0 THEN
	IF NOT Unreach_LS_Bottom THEN
		Error:=TRUE;
		ErrorID:=61;
		FB_PlcEmergencyStop();
	END_IF
ELSIF LeftTopLin.Status.Moving AND Velo_LeftTopLin<0 THEN
	IF NOT Unreach_LS_Top THEN
		Error:=TRUE;
		ErrorID:=62;
		FB_PlcEmergencyStop();
	END_IF
ELSIF RightTopLin.Status.Moving AND Velo_RightTopLin>0 THEN
	IF NOT Unreach_LS_Bottom THEN
		Error:=TRUE;
		ErrorID:=63;
		FB_PlcEmergencyStop();
	END_IF
ELSIF RightTopLin.Status.Moving AND Velo_RightTopLin<0 THEN
	IF NOT  Unreach_LS_Top THEN
		Error:=TRUE;
		ErrorID:=64;
		FB_PlcEmergencyStop();
	END_IF
ELSIF LeftBottomLin.Status.Moving AND Velo_LeftBottomLin>0 THEN
	IF NOT Unreach_LS_Bottom THEN
		Error:=TRUE;
		ErrorID:=65;
		FB_PlcEmergencyStop();
	END_IF
ELSIF LeftBottomLin.Status.Moving AND Velo_LeftBottomLin<0 THEN
	IF NOT Unreach_LS_Top THEN
		Error:=TRUE;
		ErrorID:=66;
		FB_PlcEmergencyStop();
	END_IF
ELSIF RightBottomLin.Status.Moving AND Velo_RightBottomLin>0 THEN
	IF NOT Unreach_LS_Bottom THEN
		Error:=TRUE;
		ErrorID:=67;
		FB_PlcEmergencyStop();
	END_IF
ELSIF RightBottomLin.Status.Moving AND Velo_RightBottomLin<0 THEN
	IF NOT Unreach_LS_Top THEN
		Error:=TRUE;
		ErrorID:=68;
		FB_PlcEmergencyStop();
	END_IF
END_IF
*)
(*
(******3.ÓÐÒ»¸öÏÞÎ»´¥·¢£¬ delayÊ±¼äºó£¬¼à²âÖáÊÇ·ñÔÚÍ£Ö¹×´Ì¬£¬ÈôÃ»ÓÐ£¬Emergency AND PowerOff******)
IF NOT Unreach_LS_Top OR NOT Unreach_LS_Bottom THEN
	fb_ton.IN:=TRUE;
END_IF
IF fb_ton.Q THEN
	IF LeftTopLin.Status.Moving OR RightTopLin.Status.Moving OR LeftBottomLin.Status.Moving OR RightBottomLin.Status.Moving THEN
		FB_PlcEmergencyStop();
		fb_ton.IN:=FALSE;
		Error:=TRUE;
		EStopTrig:=TRUE;
		ErrorID:=1;
		(*FB_Power_Off(Execute:=TRUE);*)
	END_IF
END_IF

(*******4.µ¥ÖáÉÏÏÂÏÞÎ»¾ùÎªFALSEÊ±£¬ÏÞÎ»´íÎó£¬Emergency*******)
IF (NOT LS_LeftTop_Top AND NOT LS_LeftTop_Bottom) OR  (NOT  LS_RightTop_Top AND NOT LS_RightTop_Bottom)
		OR (NOT LS_LeftBottom_Top AND NOT LS_LeftBottom_Bottom) OR (NOT LS_RightBottom_Top AND NOT LS_RightBottom_Bottom) THEN
	(*FB_Plc_EmergencyStop();*)
	Error:=TRUE;
	EStopTrig:=TRUE;
	ErrorID:=2;
END_IF
*)
END_ACTION

ACTION A_CheckLinearEncoder:
//
//Gap方向
//
min_UserLEProtectionGapPosition:=min_UserGapPositionNew-min_ThresholdGapSoft2LEProtection;//回程误差有0.1mm
max_UserLEProtectionGapPosition:=max_UserGapPositionNew+max_ThresholdGapSoft2LEProtection;

//如果没有使用光栅、或者光栅参数没设置好，则不检查光栅位置
IF NOT USELinearEncoder OR NOT PositionBiasDone THEN
	RETURN;
END_IF
IF Pos_LeftTopLin <=0 THEN
	ErrorID:=1101;
	Error:=TRUE;
	ErrorDescription:='Pos_LeftTopLin <=0';
	FB_PlcEmergencyStop();
	LED_Error:=TRUE;
END_IF
IF Pos_RightTopLin <=0 THEN
	ErrorID:=1102;
	Error:=TRUE;
	ErrorDescription:='Pos_RightTopLin <=0';
	FB_PlcEmergencyStop();
	LED_Error:=TRUE;
END_IF
IF Pos_LeftBottomLin <=0 THEN
	ErrorID:=1103;
	Error:=TRUE;
	ErrorDescription:='Pos_LeftBottomLin <=0';
	FB_PlcEmergencyStop();
	LED_Error:=TRUE;
END_IF
IF Pos_RightBottomLin <=0 THEN
	ErrorID:=1104;
	Error:=TRUE;
	ErrorDescription:='Pos_RightBottomLin <=0';
	FB_PlcEmergencyStop();
	LED_Error:=TRUE;
END_IF


//
IF Pos_LeftTopLin >max_UserLEProtectionGapPosition/2 THEN
	ErrorID:=1105;
	Error:=TRUE;
	ErrorDescription:='Pos_LeftTopLin >max_UserLEProtectionGapPosition/2';
	FB_PlcEmergencyStop();
	LED_Error:=TRUE;
END_IF
IF Pos_RightTopLin >max_UserLEProtectionGapPosition/2 THEN
	ErrorID:=1106;
	Error:=TRUE;
	ErrorDescription:='Pos_RightTopLin>max_UserLEProtectionGapPosition/2';
	FB_PlcEmergencyStop();
	LED_Error:=TRUE;
END_IF
IF Pos_LeftBottomLin >max_UserLEProtectionGapPosition/2 THEN
	ErrorID:=1107;
	Error:=TRUE;
	ErrorDescription:='Pos_LeftBottomLin >max_UserLEProtectionGapPosition/2';
	FB_PlcEmergencyStop();
	LED_Error:=TRUE;
END_IF
IF Pos_RightBottomLin >max_UserLEProtectionGapPosition/2 THEN
	ErrorID:=1108;
	Error:=TRUE;
	ErrorDescription:='Pos_RightBottomLin >max_UserLEProtectionGapPosition/2';
	FB_PlcEmergencyStop();
	LED_Error:=TRUE;
END_IF


IF Pos_LeftTopLin <min_UserLEProtectionGapPosition/2 THEN
	ErrorID:=1109;
	Error:=TRUE;
	ErrorDescription:='Pos_LeftTopLin <min_UserLEProtectionGapPosition/2';
	FB_PlcEmergencyStop();
	LED_Error:=TRUE;
END_IF
IF Pos_RightTopLin <min_UserLEProtectionGapPosition/2 THEN
	ErrorID:=1110;
	Error:=TRUE;
	ErrorDescription:='Pos_RightTopLin<min_UserLEProtectionGapPosition/2';
	FB_PlcEmergencyStop();
	LED_Error:=TRUE;
END_IF
IF Pos_LeftBottomLin <min_UserLEProtectionGapPosition/2 THEN
	ErrorID:=1111;
	Error:=TRUE;
	ErrorDescription:='Pos_LeftBottomLin <min_UserLEProtectionGapPosition';
	FB_PlcEmergencyStop();
	LED_Error:=TRUE;
END_IF
IF Pos_RightBottomLin <min_UserLEProtectionGapPosition/2 THEN
	ErrorID:=1112;
	Error:=TRUE;
	ErrorDescription:='Pos_RightBottomLin <min_UserLEProtectionGapPosition';
	FB_PlcEmergencyStop();
	LED_Error:=TRUE;
END_IF
END_ACTION

ACTION A_CheckMaxVelocity:
IF NOT USELinearEncoder OR NOT PositionBiasDone OR NOT IDControlReady THEN
	RETURN;
END_IF
IF NOT st_Power THEN
	RETURN;
END_IF
//Monitoring Motor and LE Position/Velocity
MaxVelocityGlobalVelocity:=MAX(UserMode.Cryogenic_ChainProtection_MoveVelocity,max_UserGapVelocityNew,
	max_UserTaperVelocityNew,UserMode.max_SS_StepVelocity,UserMode.Global_ChainProtection_MPS_MoveVelocity
	,UserMode.Global_ChainProtection_EPS_MoveVelocity);
IF 	ABS(Velo_LeftTopLin) > MaxVelocityGlobalVelocity*1.1/2 THEN
	ErrorID:=7001;
	Error:=TRUE;
	ErrorDescription:='ABS(Velo_LeftTopLin) > MaxVelocityGlobalVelocity*1.1/2';
	FB_PlcEmergencyStop();
	LED_Error:=TRUE;
END_IF
IF 	ABS(Velo_LeftTopMotor) > MaxVelocityGlobalVelocity*1.1/2 THEN
	ErrorID:=7002;
	Error:=TRUE;
	ErrorDescription:='ABS(Velo_LeftTopMotor) > MaxVelocityGlobalVelocity*1.1/2';
	FB_PlcEmergencyStop();
	LED_Error:=TRUE;
END_IF
IF 	ABS(Velo_RightTopLin) > MaxVelocityGlobalVelocity*1.1/2 THEN
	ErrorID:=7003;
	Error:=TRUE;
	ErrorDescription:='ABS(Velo_RightTopLin) > MaxVelocityGlobalVelocity*1.1/2';
	FB_PlcEmergencyStop();
	LED_Error:=TRUE;
END_IF
IF 	ABS(Velo_RightTopMotor) > MaxVelocityGlobalVelocity*1.1/2 THEN
	ErrorID:=7004;
	Error:=TRUE;
	ErrorDescription:='ABS(Velo_RightTopMotor) > MaxVelocityGlobalVelocity*1.1/2';
	FB_PlcEmergencyStop();
	LED_Error:=TRUE;
END_IF
IF 	ABS(Velo_LeftBottomLin) > MaxVelocityGlobalVelocity*1.1/2 THEN
	ErrorID:=7005;
	Error:=TRUE;
	ErrorDescription:='ABS(Velo_LeftBottomLin) > MaxVelocityGlobalVelocity*1.1/2';
	FB_PlcEmergencyStop();
	LED_Error:=TRUE;
END_IF
IF 	ABS(Velo_LeftBottomMotor) > MaxVelocityGlobalVelocity*1.1/2 THEN
	ErrorID:=7006;
	Error:=TRUE;
	ErrorDescription:='ABS(Velo_LeftBottomMotor) > MaxVelocityGlobalVelocity*1.1/2';
	FB_PlcEmergencyStop();
	LED_Error:=TRUE;
END_IF
IF 	ABS(Velo_RightBottomLin) > MaxVelocityGlobalVelocity*1.1/2 THEN
	ErrorID:=7007;
	Error:=TRUE;
	ErrorDescription:='ABS(Velo_RightBottomLin) > MaxVelocityGlobalVelocity*1.1/2';
	FB_PlcEmergencyStop();
	LED_Error:=TRUE;
END_IF
IF 	ABS(Velo_RightBottomMotor) > MaxVelocityGlobalVelocity*1.1/2 THEN
	ErrorID:=7008;
	Error:=TRUE;
	ErrorDescription:='ABS(Velo_RighBottomMotor) > MaxVelocityGlobalVelocity*1.1/2';
	FB_PlcEmergencyStop();
	LED_Error:=TRUE;
END_IF
END_ACTION

ACTION A_CryogenicCompensationMonitoring:
//没有传感器OR不是CPMU不低温补偿OR低温不到位，均不补偿
IF NOT HasTemperatureSensorOrNot OR NOT CryogenicCompensationOn THEN //OR temperatureStatus<>2 THEN
	//不补偿
	CryogenicCompensation_LeftTop:=0;
	CryogenicCompensation_RightTop:=0;
	CryogenicCompensation_LeftBottom:=0;
	CryogenicCompensation_RightBottom:=0;
ELSE
	CryogenicCompensationConditionsReady:=TRUE;//条件具备，可以低温补偿
	//检查补偿值，单轴补偿范围均在0-1内
	IF CryogenicCompensation_LeftTop>1.5 OR CryogenicCompensation_LeftTop<=0 THEN
			Error:=TRUE;
			ErrorID:=1201;
			ErrorDescription:='CryogenicCompensation_LeftTop>1 OR CryogenicCompensation_LeftTop<=0';
			FB_PlcEmergencyStop();
	END_IF
	IF CryogenicCompensation_RightTop>1.5 OR CryogenicCompensation_RightTop<=0 THEN
			Error:=TRUE;
			ErrorID:=1202;
			ErrorDescription:='CryogenicCompensation_RightTop>1 OR CryogenicCompensation_RightTop<=0';
			FB_PlcEmergencyStop();
	END_IF
	IF CryogenicCompensation_LeftBottom>1.5 OR CryogenicCompensation_LeftBottom<=0 THEN
			Error:=TRUE;
			ErrorID:=1203;
			ErrorDescription:='CryogenicCompensation_LeftBottom>1 OR CryogenicCompensation_LeftBottom<=0';
			FB_PlcEmergencyStop();
	END_IF
	IF CryogenicCompensation_RightBottom>1.5 OR CryogenicCompensation_RightBottom<=0 THEN
			Error:=TRUE;
			ErrorID:=1204;
			ErrorDescription:='CryogenicCompensation_RightBottom>1 OR CryogenicCompensation_RightBottom<=0';
			FB_PlcEmergencyStop();
	END_IF
END_IF
//若在低温补偿模式，但是温度没到低温区间，则Emergency，不允许启动
(*
IF CryogenicCompensationOn AND temperatureStatus<>2 THEN
			Error:=TRUE;
			ErrorID:=1205;
			ErrorDescription:='CryogenicCompensationOn AND temperatureStatus<>2';
			FB_PlcEmergencyStop();
END_IF
*)
//温度和模式切换连锁保护
//情况1：非低温，采用了低温模式。应当允许此间隙控制，应当执行此间隙最大运动
END_ACTION

ACTION A_GetDriverStatus:
//
//DriveMessage/Drive Number/Gear number/feedback2 direction
//
IF bReloadDriveDiagMessageAndNumber THEN
	m_GetDriveStatusState:=0;
	bReloadDriveDiagMessageAndNumber:=FALSE;
END_IF
GetDriveStatusTON(PT:=T#1S);
GetDriveStatusTON2(PT:=T#0.1S);
A_GetDriverStatusMC();
CASE m_GetDriveStatusState OF
	0:
		GetDriveStatusTON.IN:=TRUE;
		m_GetDriveStatusState:=1;
	1:
		IF GetDriveStatusTON.Q THEN
			bDriveDiagMessageAndNumber:=TRUE;
			m_GetDriveStatusState:=2;
		END_IF
	2:
		GetDriveStatusTON.IN:=FALSE;
		DriveDiagMessage_LeftTop:=fb_SoEReadDiagMessage_LeftTop.sDiagMessage.strData;
		DriveDiagMessage_RightTop:=fb_SoEReadDiagMessage_RightTop.sDiagMessage.strData;
		DriveDiagMessage_LeftBottom:=fb_SoEReadDiagMessage_LeftBottom.sDiagMessage.strData;
		DriveDiagMessage_RightBottom:=fb_SoEReadDiagMessage_RightBottom.sDiagMessage.strData;
		//
		DriveDiagNumber_LeftTop:=FB_SoEReadDiagNumber_LeftTop.iDiagNumber;
		DriveDiagNumber_RightTop:=FB_SoEReadDiagNumber_RightTop.iDiagNumber;
		DriveDiagNumber_LeftBottom:=FB_SoEReadDiagNumber_LeftBottom.iDiagNumber;
		DriveDiagNumber_RightBottom:=FB_SoEReadDiagNumber_RightBottom.iDiagNumber;
		//
		GearNumeratorGet_LeftTop:=st_p182_LeftTop.Feedback_2_geat_numerator;
		GearNumeratorGet_RightTop:=st_p182_RightTop.Feedback_2_geat_numerator;
		GearNumeratorGet_LeftBottom:=st_p182_LeftBottom.Feedback_2_geat_numerator;
		GearNumeratorGet_RightBottom:=st_p182_RightBottom.Feedback_2_geat_numerator;
		//
		GearDenominatorGet_LeftTop:=st_p183_LeftTop.Feedback_2_geat_denominator;
		GearDenominatorGet_RightTop:=st_p183_RightTop.Feedback_2_geat_denominator;
		GearDenominatorGet_LeftBottom:=st_p183_LeftBottom.Feedback_2_geat_denominator;
		GearDenominatorGet_RightBottom:=st_p183_RightBottom.Feedback_2_geat_denominator;
		//
		Feedback2directionGet_LeftTop:=st_p180_LeftTop.Feedback_direction;
		Feedback2directionGet_RightTop:=st_p180_RightTop.Feedback_direction;
		Feedback2directionGet_LeftBottom:=st_p180_LeftBottom.Feedback_direction;
		Feedback2directionGet_RightBottom:=st_p180_RightBottom.Feedback_direction;
		//
		IF 	NOT fb_SoEReadDiagMessage_LeftTop.bBusy
			AND NOT fb_SoEReadDiagMessage_RightTop.bBusy
			AND NOT fb_SoEReadDiagMessage_LeftBottom.bBusy
			AND NOT fb_SoEReadDiagMessage_RightBottom.bBusy 
			AND NOT FB_SoEReadDiagNumber_LeftTop.bBusy
			AND NOT  FB_SoEReadDiagNumber_RightTop.bBusy
			AND NOT FB_SoEReadDiagNumber_LeftBottom.bBusy
			AND NOT FB_SoEReadDiagNumber_RightBottom.bBusy 
			AND NOT FB_SoERead_GearNumerator_LeftTop.bBusy 
			AND NOT FB_SoERead_GearNumerator_RightTop.bBusy 
			AND NOT FB_SoERead_GearNumerator_LeftBottom.bBusy 
			AND NOT FB_SoERead_GearNumerator_RightBottom.bBusy 
			AND NOT FB_SoERead_GearDenominator_LeftTop.bBusy 
			AND NOT FB_SoERead_GearDenominator_RightTop.bBusy 
			AND NOT FB_SoERead_GearDenominator_LeftBottom.bBusy 
			AND NOT FB_SoERead_GearDenominator_RightBottom.bBusy 
			AND NOT FB_SoERead_Feedback2direction_LeftTop.bBusy 
			AND NOT FB_SoERead_Feedback2direction_RightTop.bBusy 
			AND NOT FB_SoERead_Feedback2direction_LeftBottom.bBusy 
			AND NOT FB_SoERead_Feedback2direction_RightBottom.bBusy	THEN
				GetDriveStatusTON2.IN:=TRUE;
				IF GetDriveStatusTON2.Q THEN
					m_GetDriveStatusState:=88;
				END_IF
		END_IF
		IF 	fb_SoEReadDiagMessage_LeftTop.bError
			OR fb_SoEReadDiagMessage_RightTop.bError
			OR fb_SoEReadDiagMessage_LeftBottom.bError
			OR fb_SoEReadDiagMessage_RightBottom.bError
			OR FB_SoEReadDiagNumber_LeftTop.bError
			OR FB_SoEReadDiagNumber_RightTop.bError
			OR FB_SoEReadDiagNumber_LeftBottom.bError
			OR FB_SoEReadDiagNumber_RightBottom.bError 
			OR FB_SoERead_GearNumerator_LeftTop.bError 
			OR FB_SoERead_GearNumerator_RightTop.bError 
			OR FB_SoERead_GearNumerator_LeftBottom.bError 
			OR FB_SoERead_GearNumerator_RightBottom.bError 
			OR FB_SoERead_GearDenominator_LeftTop.bError 
			OR FB_SoERead_GearDenominator_RightTop.bError 
			OR FB_SoERead_GearDenominator_LeftBottom.bError 
			OR FB_SoERead_GearDenominator_RightBottom.bError 
			OR FB_SoERead_Feedback2direction_LeftTop.bError 
			OR FB_SoERead_Feedback2direction_RightTop.bError 
			OR FB_SoERead_Feedback2direction_LeftBottom.bError 
			OR FB_SoERead_Feedback2direction_RightBottom.bError 
		THEN
			m_GetDriveStatusState:=-100;
		END_IF
		
	88:
		bDriveDiagMessageAndNumber:=FALSE;
		A_GetDriverStatusMC();
		GetDriveStatusStateDone:=TRUE;
		GetDriveStatusStateError:=FALSE;
		//
		(*Drive Status*)
		//D012, Axis state machine: Control and power section ready,53266
		IF DriveDiagNumber_LeftTop=16#D012 AND DriveDiagNumber_RightTop=16#D012
			AND DriveDiagNumber_LeftBottom=16#D012 AND DriveDiagNumber_RightBottom=16#D012 THEN
			DriveStatus:=1;
		//D013, Axis state machine: Axis in operation,53267
		ELSIF DriveDiagNumber_LeftTop=16#D013 AND DriveDiagNumber_RightTop=16#D013
			AND DriveDiagNumber_LeftBottom=16#D013 AND DriveDiagNumber_RightBottom=16#D013 THEN
			DriveStatus:=2;
		//D014，Axis state machine: Axis halt.53266和53267中间会经历这么一个状态，算正常状态
		ELSIF DriveDiagNumber_LeftTop=16#D014 AND DriveDiagNumber_RightTop=16#D014
			AND DriveDiagNumber_LeftBottom=16#D014 AND DriveDiagNumber_RightBottom=16#D014 THEN
			DriveStatus:=3;
		ELSE
			DriveStatus:=0;
		END_IF
		//
		//
		//	//check statusGet and status configured
		IF 	GearNumeratorGet_LeftTop<>GearNumeratorConfigured_LeftTop 
			OR GearNumeratorGet_RightTop<>GearNumeratorConfigured_RightTop
			OR GearNumeratorGet_LeftBottom<>GearNumeratorConfigured_LeftBottom 
			OR GearNumeratorGet_RightBottom<>GearNumeratorConfigured_RightBottom
			OR GearDenominatorGet_LeftTop<>GearDenominatorConfigured_LeftTop 
			OR GearDenominatorGet_RightTop<>GearDenominatorConfigured_RightTop
			OR GearDenominatorGet_LeftBottom<>GearDenominatorConfigured_LeftBottom 
			OR GearDenominatorGet_RightBottom<>GearDenominatorConfigured_RightBottom	THEN
				bDriveDiagMessageAndNumber:=FALSE;
				A_GetDriverStatusMC();
				GetDriveStatusStateDone:=FALSE;
				GetDriveStatusStateError:=TRUE;
				Error:=TRUE;
				ErrorId:=1302;
				ErrorDescription:='gearParameters Error';
				Plc_EmergencyStop:=FALSE;
		END_IF
		IF USELinearEncoder THEN
			IF Feedback2directionGet_LeftTop<>Feedback2directionConfigured_LeftTop 
				OR Feedback2directionGet_RightTop<>Feedback2directionConfigured_RightTop
				OR Feedback2directionGet_LeftBottom<>Feedback2directionConfigured_LeftBottom 
				OR Feedback2directionGet_RightBottom<Feedback2directionConfigured_RightBottom THEN
					bDriveDiagMessageAndNumber:=FALSE;
					A_GetDriverStatusMC();
					GetDriveStatusStateDone:=FALSE;
					GetDriveStatusStateError:=TRUE;
					Error:=TRUE;
					ErrorId:=1303;
					ErrorDescription:='fb2direction Error';
					Plc_EmergencyStop:=FALSE;	
			END_IF				
		END_IF
		m_GetDriveStatusState:=0;
	-100:
		bDriveDiagMessageAndNumber:=FALSE;
		A_GetDriverStatusMC();
		GetDriveStatusStateDone:=FALSE;
		GetDriveStatusStateError:=TRUE;
		Error:=TRUE;
		ErrorId:=1301;
		ErrorDescription:='GetDriveStatusStateError';
END_CASE
END_ACTION

ACTION A_GetDriverStatusMC:
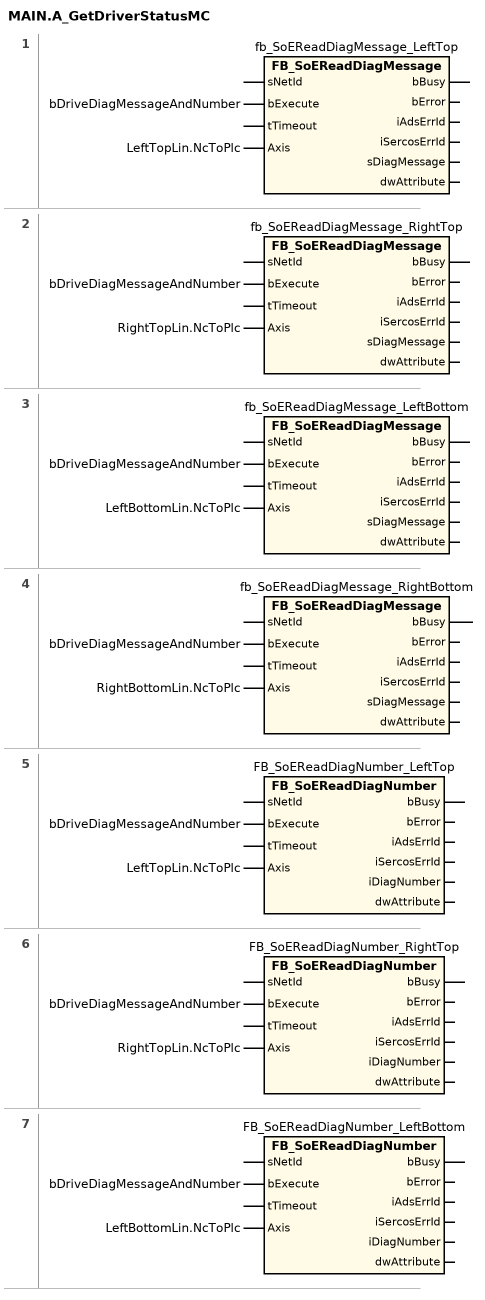
// NETWORK 1
fb_SoEReadDiagMessage_LeftTop(bExecute := bDriveDiagMessageAndNumber, Axis := LeftTopLin.NcToPlc); // FB_SoEReadDiagMessage

// NETWORK 2
fb_SoEReadDiagMessage_RightTop(bExecute := bDriveDiagMessageAndNumber, Axis := RightTopLin.NcToPlc); // FB_SoEReadDiagMessage

// NETWORK 3
fb_SoEReadDiagMessage_LeftBottom(bExecute := bDriveDiagMessageAndNumber, Axis := LeftBottomLin.NcToPlc); // FB_SoEReadDiagMessage

// NETWORK 4
fb_SoEReadDiagMessage_RightBottom(bExecute := bDriveDiagMessageAndNumber, Axis := RightBottomLin.NcToPlc); // FB_SoEReadDiagMessage

// NETWORK 5
FB_SoEReadDiagNumber_LeftTop(bExecute := bDriveDiagMessageAndNumber, Axis := LeftTopLin.NcToPlc); // FB_SoEReadDiagNumber

// NETWORK 6
FB_SoEReadDiagNumber_RightTop(bExecute := bDriveDiagMessageAndNumber, Axis := RightTopLin.NcToPlc); // FB_SoEReadDiagNumber

// NETWORK 7
FB_SoEReadDiagNumber_LeftBottom(bExecute := bDriveDiagMessageAndNumber, Axis := LeftBottomLin.NcToPlc); // FB_SoEReadDiagNumber

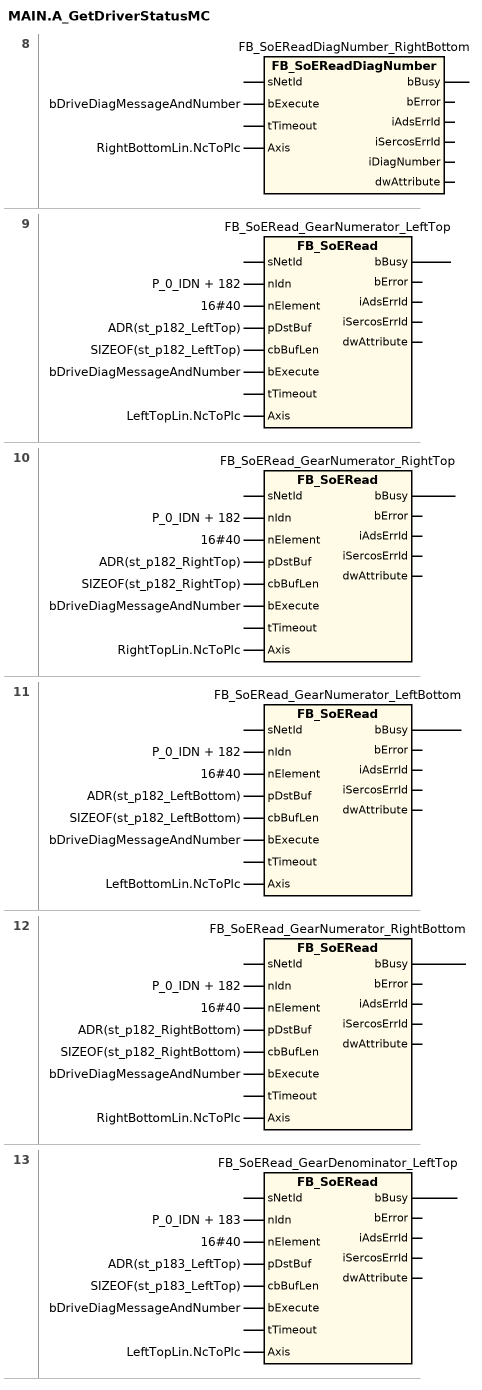
// NETWORK 8
FB_SoEReadDiagNumber_RightBottom(bExecute := bDriveDiagMessageAndNumber, Axis := RightBottomLin.NcToPlc); // FB_SoEReadDiagNumber

// NETWORK 9
FB_SoERead_GearNumerator_LeftTop(
    nIdn := P_0_IDN + 182,
    nElement := 16#40,
    pDstBuf := ADR(st_p182_LeftTop),
    cbBufLen := SIZEOF(st_p182_LeftTop),
    bExecute := bDriveDiagMessageAndNumber,
    Axis := LeftTopLin.NcToPlc); // FB_SoERead

// NETWORK 10
FB_SoERead_GearNumerator_RightTop(
    nIdn := P_0_IDN + 182,
    nElement := 16#40,
    pDstBuf := ADR(st_p182_RightTop),
    cbBufLen := SIZEOF(st_p182_RightTop),
    bExecute := bDriveDiagMessageAndNumber,
    Axis := RightTopLin.NcToPlc); // FB_SoERead

// NETWORK 11
FB_SoERead_GearNumerator_LeftBottom(
    nIdn := P_0_IDN + 182,
    nElement := 16#40,
    pDstBuf := ADR(st_p182_LeftBottom),
    cbBufLen := SIZEOF(st_p182_LeftBottom),
    bExecute := bDriveDiagMessageAndNumber,
    Axis := LeftBottomLin.NcToPlc); // FB_SoERead

// NETWORK 12
FB_SoERead_GearNumerator_RightBottom(
    nIdn := P_0_IDN + 182,
    nElement := 16#40,
    pDstBuf := ADR(st_p182_RightBottom),
    cbBufLen := SIZEOF(st_p182_RightBottom),
    bExecute := bDriveDiagMessageAndNumber,
    Axis := RightBottomLin.NcToPlc); // FB_SoERead

// NETWORK 13
FB_SoERead_GearDenominator_LeftTop(
    nIdn := P_0_IDN + 183,
    nElement := 16#40,
    pDstBuf := ADR(st_p183_LeftTop),
    cbBufLen := SIZEOF(st_p183_LeftTop),
    bExecute := bDriveDiagMessageAndNumber,
    Axis := LeftTopLin.NcToPlc); // FB_SoERead

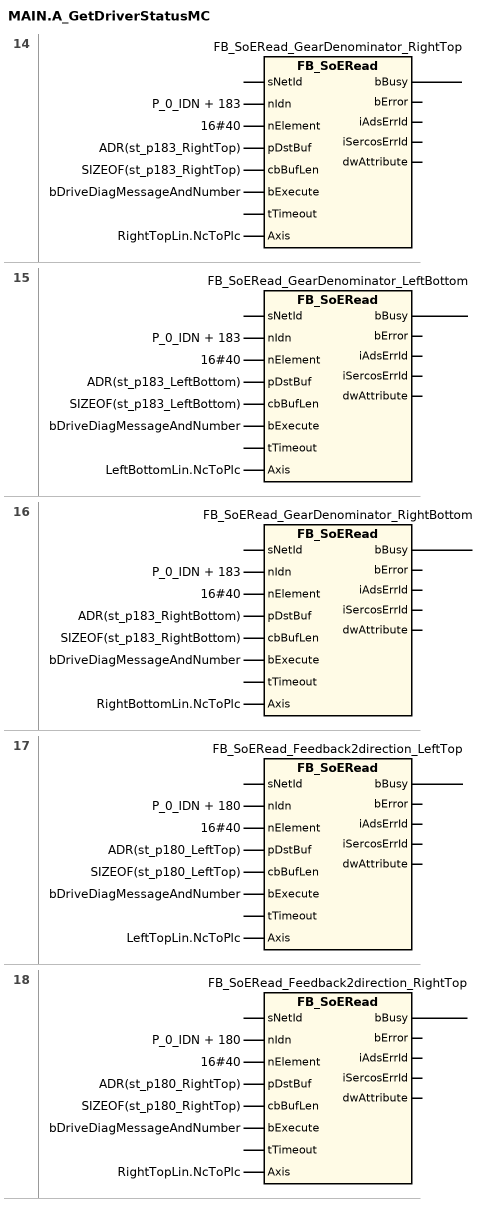
// NETWORK 14
FB_SoERead_GearDenominator_RightTop(
    nIdn := P_0_IDN + 183,
    nElement := 16#40,
    pDstBuf := ADR(st_p183_RightTop),
    cbBufLen := SIZEOF(st_p183_RightTop),
    bExecute := bDriveDiagMessageAndNumber,
    Axis := RightTopLin.NcToPlc); // FB_SoERead

// NETWORK 15
FB_SoERead_GearDenominator_LeftBottom(
    nIdn := P_0_IDN + 183,
    nElement := 16#40,
    pDstBuf := ADR(st_p183_LeftBottom),
    cbBufLen := SIZEOF(st_p183_LeftBottom),
    bExecute := bDriveDiagMessageAndNumber,
    Axis := LeftBottomLin.NcToPlc); // FB_SoERead

// NETWORK 16
FB_SoERead_GearDenominator_RightBottom(
    nIdn := P_0_IDN + 183,
    nElement := 16#40,
    pDstBuf := ADR(st_p183_RightBottom),
    cbBufLen := SIZEOF(st_p183_RightBottom),
    bExecute := bDriveDiagMessageAndNumber,
    Axis := RightBottomLin.NcToPlc); // FB_SoERead

// NETWORK 17
FB_SoERead_Feedback2direction_LeftTop(
    nIdn := P_0_IDN + 180,
    nElement := 16#40,
    pDstBuf := ADR(st_p180_LeftTop),
    cbBufLen := SIZEOF(st_p180_LeftTop),
    bExecute := bDriveDiagMessageAndNumber,
    Axis := LeftTopLin.NcToPlc); // FB_SoERead

// NETWORK 18
FB_SoERead_Feedback2direction_RightTop(
    nIdn := P_0_IDN + 180,
    nElement := 16#40,
    pDstBuf := ADR(st_p180_RightTop),
    cbBufLen := SIZEOF(st_p180_RightTop),
    bExecute := bDriveDiagMessageAndNumber,
    Axis := RightTopLin.NcToPlc); // FB_SoERead

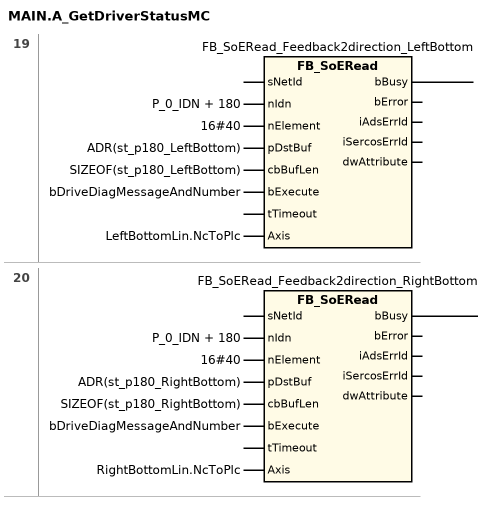
// NETWORK 19
FB_SoERead_Feedback2direction_LeftBottom(
    nIdn := P_0_IDN + 180,
    nElement := 16#40,
    pDstBuf := ADR(st_p180_LeftBottom),
    cbBufLen := SIZEOF(st_p180_LeftBottom),
    bExecute := bDriveDiagMessageAndNumber,
    Axis := LeftBottomLin.NcToPlc); // FB_SoERead

// NETWORK 20
FB_SoERead_Feedback2direction_RightBottom(
    nIdn := P_0_IDN + 180,
    nElement := 16#40,
    pDstBuf := ADR(st_p180_RightBottom),
    cbBufLen := SIZEOF(st_p180_RightBottom),
    bExecute := bDriveDiagMessageAndNumber,
    Axis := RightBottomLin.NcToPlc); // FB_SoERead
END_ACTION

ACTION A_GetMotorTemperature:
MotorTemperature_LeftTop:=UINT_TO_LREAL(MotorTemperature[0])/10;
MotorTemperature_RightTop:=UINT_TO_LREAL(MotorTemperature[1])/10;
MotorTemperature_LeftBottom:=UINT_TO_LREAL(MotorTemperature[2])/10;
MotorTemperature_RightBottom:=UINT_TO_LREAL(MotorTemperature[3])/10;
END_ACTION

ACTION A_GetScaleFactor:
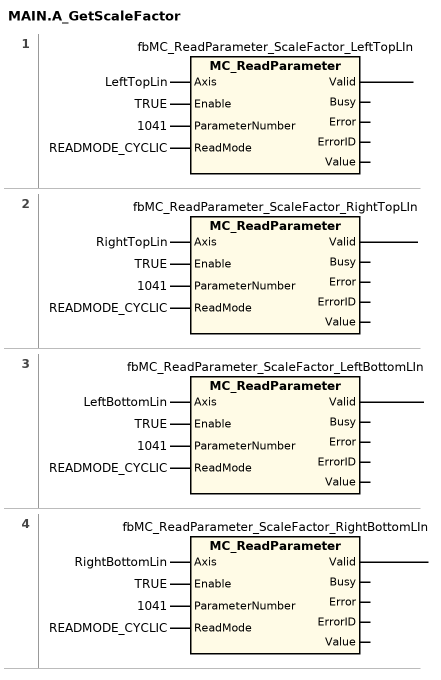
// NETWORK 1
fbMC_ReadParameter_ScaleFactor_LeftTopLIn(
    Axis := LeftTopLin,
    Enable := TRUE,
    ParameterNumber := 1041,
    ReadMode := READMODE_CYCLIC); // MC_ReadParameter

// NETWORK 2
fbMC_ReadParameter_ScaleFactor_RightTopLIn(
    Axis := RightTopLin,
    Enable := TRUE,
    ParameterNumber := 1041,
    ReadMode := READMODE_CYCLIC); // MC_ReadParameter

// NETWORK 3
fbMC_ReadParameter_ScaleFactor_LeftBottomLIn(
    Axis := LeftBottomLin,
    Enable := TRUE,
    ParameterNumber := 1041,
    ReadMode := READMODE_CYCLIC); // MC_ReadParameter

// NETWORK 4
fbMC_ReadParameter_ScaleFactor_RightBottomLIn(
    Axis := RightBottomLin,
    Enable := TRUE,
    ParameterNumber := 1041,
    ReadMode := READMODE_CYCLIC); // MC_ReadParameter
END_ACTION

ACTION A_GetTemperatureSensorsData:
IF TempSensorHardware=1 THEN//from profibus,lakeshore 240-8P
	//sensor_1
	dut_sensor_datas_1.data_byte[3]:=Sensor_Reading_1[0];
	dut_sensor_datas_1.data_byte[2]:=Sensor_Reading_1[1];
	dut_sensor_datas_1.data_byte[1]:=Sensor_Reading_1[2];
	dut_sensor_datas_1.data_byte[0]:=Sensor_Reading_1[3];
	TemperatureSensors_1:=DINT_TO_LREAL(LREAL_TO_DINT(dut_sensor_datas_1.data_lreal*100))/100;
	//sensor_2
	dut_sensor_datas_2.data_byte[3]:=Sensor_Reading_2[0];
	dut_sensor_datas_2.data_byte[2]:=Sensor_Reading_2[1];
	dut_sensor_datas_2.data_byte[1]:=Sensor_Reading_2[2];
	dut_sensor_datas_2.data_byte[0]:=Sensor_Reading_2[3];
	TemperatureSensors_2:=DINT_TO_LREAL(LREAL_TO_DINT(dut_sensor_datas_2.data_lreal*100))/100;
	//sensor_3
	dut_sensor_datas_3.data_byte[3]:=Sensor_Reading_3[0];
	dut_sensor_datas_3.data_byte[2]:=Sensor_Reading_3[1];
	dut_sensor_datas_3.data_byte[1]:=Sensor_Reading_3[2];
	dut_sensor_datas_3.data_byte[0]:=Sensor_Reading_3[3];
	TemperatureSensors_3:=DINT_TO_LREAL(LREAL_TO_DINT(dut_sensor_datas_3.data_lreal*100))/100;
	//sensor_4
	dut_sensor_datas_4.data_byte[3]:=Sensor_Reading_4[0];
	dut_sensor_datas_4.data_byte[2]:=Sensor_Reading_4[1];
	dut_sensor_datas_4.data_byte[1]:=Sensor_Reading_4[2];
	dut_sensor_datas_4.data_byte[0]:=Sensor_Reading_4[3];
	TemperatureSensors_4:=DINT_TO_LREAL(LREAL_TO_DINT(dut_sensor_datas_4.data_lreal*100))/100;
	//sensor_5
	dut_sensor_datas_5.data_byte[3]:=Sensor_Reading_5[0];
	dut_sensor_datas_5.data_byte[2]:=Sensor_Reading_5[1];
	dut_sensor_datas_5.data_byte[1]:=Sensor_Reading_5[2];
	dut_sensor_datas_5.data_byte[0]:=Sensor_Reading_5[3];
	TemperatureSensors_5:=DINT_TO_LREAL(LREAL_TO_DINT(dut_sensor_datas_5.data_lreal*100))/100;
	//sensor_6
	dut_sensor_datas_6.data_byte[3]:=Sensor_Reading_6[0];
	dut_sensor_datas_6.data_byte[2]:=Sensor_Reading_6[1];
	dut_sensor_datas_6.data_byte[1]:=Sensor_Reading_6[2];
	dut_sensor_datas_6.data_byte[0]:=Sensor_Reading_6[3];
	TemperatureSensors_6:=DINT_TO_LREAL(LREAL_TO_DINT(dut_sensor_datas_6.data_lreal*100))/100;
	//sensor_7
	dut_sensor_datas_7.data_byte[3]:=Sensor_Reading_7[0];
	dut_sensor_datas_7.data_byte[2]:=Sensor_Reading_7[1];
	dut_sensor_datas_7.data_byte[1]:=Sensor_Reading_7[2];
	dut_sensor_datas_7.data_byte[0]:=Sensor_Reading_7[3];
	TemperatureSensors_7:=DINT_TO_LREAL(LREAL_TO_DINT(dut_sensor_datas_7.data_lreal*100))/100;
	//sensor_8
	dut_sensor_datas_8.data_byte[3]:=Sensor_Reading_8[0];
	dut_sensor_datas_8.data_byte[2]:=Sensor_Reading_8[1];
	dut_sensor_datas_8.data_byte[1]:=Sensor_Reading_8[2];
	dut_sensor_datas_8.data_byte[0]:=Sensor_Reading_8[3];
	TemperatureSensors_8:=DINT_TO_LREAL(LREAL_TO_DINT(dut_sensor_datas_8.data_lreal*100))/100;
END_IF
IF TempSensorHardware=2 THEN//from BECKHOFF EL3202
	TemperatureSensors_1:=INT_TO_LREAL(EL3202_Reading[0])/100;
	TemperatureSensors_2:=INT_TO_LREAL(EL3202_Reading[1])/100;
	TemperatureSensors_3:=INT_TO_LREAL(EL3202_Reading[2])/100;
	TemperatureSensors_4:=INT_TO_LREAL(EL3202_Reading[3])/100;
	TemperatureSensors_5:=INT_TO_LREAL(EL3202_Reading[4])/100;
	TemperatureSensors_6:=INT_TO_LREAL(EL3202_Reading[5])/100;
	TemperatureSensors_7:=INT_TO_LREAL(EL3202_Reading[6])/100;
	TemperatureSensors_8:=INT_TO_LREAL(EL3202_Reading[7])/100;
END_IF
//计算temperature_gradient
temperature_gradient_2_To_1:=ABS(TemperatureSensors_2-TemperatureSensors_1);
temperature_gradient_3_To_2:=ABS(TemperatureSensors_3-TemperatureSensors_2);
temperature_gradient_5_To_4:=ABS(TemperatureSensors_5-TemperatureSensors_4);
temperature_gradient_6_To_5:=ABS(TemperatureSensors_6-TemperatureSensors_5);
temperature_gradient_max:=DINT_TO_LREAL(LREAL_TO_DINT(MAX(temperature_gradient_2_To_1,temperature_gradient_3_To_2,
							temperature_gradient_5_To_4,temperature_gradient_6_To_5)*100))/100;
//计算大梁上的温度平均值
temperature_average:=DINT_TO_LREAL(LREAL_TO_DINT((TemperatureSensors_1+TemperatureSensors_2+TemperatureSensors_3+TemperatureSensors_4
					+TemperatureSensors_5+TemperatureSensors_6)/6*100))/100;
					

//传感器温度状态：0：有传感器度数错误；1:常温；2:低温；3:常温和低温中间态
IF TemperatureSensors_1=0 OR TemperatureSensors_2=0 OR TemperatureSensors_3=0 
	OR TemperatureSensors_4=0 OR TemperatureSensors_5=0 OR TemperatureSensors_6=0 THEN	
	temperatureStatus:=0;//有传感器读数错误
ELSIF TemperatureSensors_1>=RoomTemperatureThreshold AND TemperatureSensors_2>=RoomTemperatureThreshold AND TemperatureSensors_3>=RoomTemperatureThreshold
	AND TemperatureSensors_4>=RoomTemperatureThreshold AND TemperatureSensors_5>=RoomTemperatureThreshold AND TemperatureSensors_6>=RoomTemperatureThreshold THEN	
	temperatureStatus:=1;//常温
	InCryogenicOrNot:=FALSE;
ELSIF TemperatureSensors_1<=CryogenicTemperatureThreshold AND TemperatureSensors_1>70
	AND TemperatureSensors_2<=CryogenicTemperatureThreshold  AND TemperatureSensors_2>70
	AND TemperatureSensors_3<=CryogenicTemperatureThreshold  AND TemperatureSensors_3>70
	AND TemperatureSensors_4<=CryogenicTemperatureThreshold   AND TemperatureSensors_4>70
	AND TemperatureSensors_5<=CryogenicTemperatureThreshold  AND TemperatureSensors_5>70
	AND TemperatureSensors_6<=CryogenicTemperatureThreshold   AND TemperatureSensors_6>70 THEN	
	temperatureStatus:=2;//低温
	InCryogenicOrNot:=TRUE;
ELSE
	temperatureStatus:=3;//常温和低温中间
	InCryogenicOrNot:=FALSE;
END_IF
							
//
//high temperature
//		
IF TempSensorHardware=1 THEN//from profibus,lakeshore 240-8P		
	//sensor_h1
	dut_sensor_datas_h1.data_byte[3]:=Sensor_Reading_h1[0];
	dut_sensor_datas_h1.data_byte[2]:=Sensor_Reading_h1[1];
	dut_sensor_datas_h1.data_byte[1]:=Sensor_Reading_h1[2];
	dut_sensor_datas_h1.data_byte[0]:=Sensor_Reading_h1[3];
	TemperatureSensors_h1:=DINT_TO_LREAL(LREAL_TO_DINT(dut_sensor_datas_h1.data_lreal*100))/100;
	//sensor_h2
	dut_sensor_datas_h2.data_byte[3]:=Sensor_Reading_h2[0];
	dut_sensor_datas_h2.data_byte[2]:=Sensor_Reading_h2[1];
	dut_sensor_datas_h2.data_byte[1]:=Sensor_Reading_h2[2];
	dut_sensor_datas_h2.data_byte[0]:=Sensor_Reading_h2[3];
	TemperatureSensors_h2:=DINT_TO_LREAL(LREAL_TO_DINT(dut_sensor_datas_h2.data_lreal*100))/100;
	//sensor_h3
	dut_sensor_datas_h3.data_byte[3]:=Sensor_Reading_h3[0];
	dut_sensor_datas_h3.data_byte[2]:=Sensor_Reading_h3[1];
	dut_sensor_datas_h3.data_byte[1]:=Sensor_Reading_h3[2];
	dut_sensor_datas_h3.data_byte[0]:=Sensor_Reading_h3[3];
	TemperatureSensors_h3:=DINT_TO_LREAL(LREAL_TO_DINT(dut_sensor_datas_h3.data_lreal*100))/100;
	//sensor_h4
	dut_sensor_datas_h4.data_byte[3]:=Sensor_Reading_h4[0];
	dut_sensor_datas_h4.data_byte[2]:=Sensor_Reading_h4[1];
	dut_sensor_datas_h4.data_byte[1]:=Sensor_Reading_h4[2];
	dut_sensor_datas_h4.data_byte[0]:=Sensor_Reading_h4[3];
	TemperatureSensors_h4:=DINT_TO_LREAL(LREAL_TO_DINT(dut_sensor_datas_h4.data_lreal*100))/100;
	//sensor_h5
	dut_sensor_datas_h5.data_byte[3]:=Sensor_Reading_h5[0];
	dut_sensor_datas_h5.data_byte[2]:=Sensor_Reading_h5[1];
	dut_sensor_datas_h5.data_byte[1]:=Sensor_Reading_h5[2];
	dut_sensor_datas_h5.data_byte[0]:=Sensor_Reading_h5[3];
	TemperatureSensors_h5:=DINT_TO_LREAL(LREAL_TO_DINT(dut_sensor_datas_h5.data_lreal*100))/100;
	//sensor_h6
	dut_sensor_datas_h6.data_byte[3]:=Sensor_Reading_h6[0];
	dut_sensor_datas_h6.data_byte[2]:=Sensor_Reading_h6[1];
	dut_sensor_datas_h6.data_byte[1]:=Sensor_Reading_h6[2];
	dut_sensor_datas_h6.data_byte[0]:=Sensor_Reading_h6[3];
	TemperatureSensors_h6:=DINT_TO_LREAL(LREAL_TO_DINT(dut_sensor_datas_h6.data_lreal*100))/100;
	//sensor_h7
	dut_sensor_datas_h7.data_byte[3]:=Sensor_Reading_h7[0];
	dut_sensor_datas_h7.data_byte[2]:=Sensor_Reading_h7[1];
	dut_sensor_datas_h7.data_byte[1]:=Sensor_Reading_h7[2];
	dut_sensor_datas_h7.data_byte[0]:=Sensor_Reading_h7[3];
	TemperatureSensors_h7:=DINT_TO_LREAL(LREAL_TO_DINT(dut_sensor_datas_h7.data_lreal*100))/100;
	//sensor_h8
	dut_sensor_datas_h8.data_byte[3]:=Sensor_Reading_h8[0];
	dut_sensor_datas_h8.data_byte[2]:=Sensor_Reading_h8[1];
	dut_sensor_datas_h8.data_byte[1]:=Sensor_Reading_h8[2];
	dut_sensor_datas_h8.data_byte[0]:=Sensor_Reading_h8[3];
	TemperatureSensors_h8:=DINT_TO_LREAL(LREAL_TO_DINT(dut_sensor_datas_h8.data_lreal*100))/100;
END_IF
IF TempSensorHardware=2 THEN//from BECKHOFF EL3202
	TemperatureSensors_h1:=INT_TO_LREAL(EL3202_hReading[0])/100;
	TemperatureSensors_h2:=INT_TO_LREAL(EL3202_hReading[1])/100;
	TemperatureSensors_h3:=INT_TO_LREAL(EL3202_hReading[2])/100;
	TemperatureSensors_h4:=INT_TO_LREAL(EL3202_hReading[3])/100;
	TemperatureSensors_h5:=INT_TO_LREAL(EL3202_hReading[4])/100;
	TemperatureSensors_h6:=INT_TO_LREAL(EL3202_hReading[5])/100;
	TemperatureSensors_h7:=INT_TO_LREAL(EL3202_hReading[6])/100;
	TemperatureSensors_h8:=INT_TO_LREAL(EL3202_hReading[7])/100;
END_IF
//计算temperature_gradient
temperature_gradient_h2_To_h1:=ABS(TemperatureSensors_h2-TemperatureSensors_h1);
temperature_gradient_h3_To_h2:=ABS(TemperatureSensors_h3-TemperatureSensors_h2);
temperature_gradient_h5_To_h4:=ABS(TemperatureSensors_h5-TemperatureSensors_h4);
temperature_gradient_h6_To_h5:=ABS(TemperatureSensors_h6-TemperatureSensors_h5);
temperature_gradient_maxh:=DINT_TO_LREAL(LREAL_TO_DINT(MAX(temperature_gradient_h2_To_h1,temperature_gradient_h3_To_h2,
							temperature_gradient_h5_To_h4,temperature_gradient_h6_To_h5)*100))/100;
//计算大梁上的温度平均值
temperature_averageh:=DINT_TO_LREAL(LREAL_TO_DINT((TemperatureSensors_h1+TemperatureSensors_h2+TemperatureSensors_h3+TemperatureSensors_h4
					+TemperatureSensors_h5+TemperatureSensors_h6)/6*100))/100;
END_ACTION

ACTION A_InitAxisParameters:
(*LinearEncoder Pos Velo Lagdistance status get*)
	//Position
	Pos_LeftTopLin:=DINT_TO_LREAL(LREAL_TO_DINT(LeftTopLin.NcToPlc.ActPos*100000))/100000;
	Pos_RightTopLin:=DINT_TO_LREAL(LREAL_TO_DINT(RightTopLin.NcToPlc.ActPos*100000))/100000;
	Pos_LeftBottomLin:=DINT_TO_LREAL(LREAL_TO_DINT(LeftBottomLin.NcToPlc.ActPos*100000))/100000;
	Pos_RightBottomLin:=DINT_TO_LREAL(LREAL_TO_DINT(RightBottomLin.NcToPlc.ActPos*100000))/100000;
	//Moving status
	moveStatusLeftTop:=LeftTopLin.Status.Moving;
	moveStatusRightTop:=RightTopLin.Status.Moving;
	moveStatusLeftBottom:=LeftBottomLin.Status.Moving;
	moveStatusRightBottom:=RightBottomLin.Status.Moving;
	moveStatusAllAxis:=moveStatusLeftTop AND moveStatusRightTop AND moveStatusLeftBottom AND moveStatusRightBottom;
	moveStatusAnyAxis:=moveStatusLeftTop OR moveStatusRightTop OR moveStatusLeftBottom OR moveStatusRightBottom;
	//Velocity
	Velo_LeftTopLin:=DINT_TO_LREAL(LREAL_TO_DINT(LeftTopLin.NcToPlc.ActVelo*100000))/100000;
	Velo_RightTopLin:=DINT_TO_LREAL(LREAL_TO_DINT(RightTopLin.NcToPlc.ActVelo*100000))/100000;
	Velo_LeftBottomLin:=DINT_TO_LREAL(LREAL_TO_DINT(LeftBottomLin.NcToPlc.ActVelo*100000))/100000;
	Velo_RightBottomLin:=DINT_TO_LREAL(LREAL_TO_DINT(RightBottomLin.NcToPlc.ActVelo*100000))/100000;
	//LagDistance
	PosDiff_LeftTopLin_actual:=DINT_TO_LREAL(LREAL_TO_DINT(LeftTopLin.NcToPlc.PosDiff*100000))/100000;
	PosDiff_RightTopLin_actual:=DINT_TO_LREAL(LREAL_TO_DINT(RightTopLin.NcToPlc.PosDiff*100000))/100000;
	PosDiff_LeftBottomLin_actual:=DINT_TO_LREAL(LREAL_TO_DINT(LeftBottomLin.NcToPlc.PosDiff*100000))/100000;
	PosDiff_RightBottomLin_actual:=DINT_TO_LREAL(LREAL_TO_DINT(RightBottomLin.NcToPlc.PosDiff*100000))/100000;
	//Torque
	Torque_LeftTopLin:=DINT_TO_LREAL(LREAL_TO_DINT(LeftTopLin.NcToPlc.ActTorque*100000))/100000;
	Torque_RightTopLin:=DINT_TO_LREAL(LREAL_TO_DINT(RightTopLin.NcToPlc.ActTorque*100000))/100000;
	Torque_LeftBottomLin:=DINT_TO_LREAL(LREAL_TO_DINT(LeftBottomLin.NcToPlc.ActTorque*100000))/100000;
	Torque_RightBottomLin:=DINT_TO_LREAL(LREAL_TO_DINT(RightBottomLin.NcToPlc.ActTorque*100000))/100000;

	LeftTopLin.ReadStatus();
	RightTopLin.ReadStatus();
	LeftBottomLin.ReadStatus();
	RightBottomLin.ReadStatus();
	
	(*Motor Pos Velo Lagdistance status get*)
	//Position
	Pos_LeftTopMotor:=DINT_TO_LREAL(LREAL_TO_DINT(LeftTopMotor.NcToPlc.ActPos*100000))/100000;
	Pos_RightTopMotor:=DINT_TO_LREAL(LREAL_TO_DINT(RightTopMotor.NcToPlc.ActPos*100000))/100000;
	Pos_LeftBottomMotor:=DINT_TO_LREAL(LREAL_TO_DINT(LeftBottomMotor.NcToPlc.ActPos*100000))/100000;
	Pos_RightBottomMotor:=DINT_TO_LREAL(LREAL_TO_DINT(RightBottomMotor.NcToPlc.ActPos*100000))/100000;
	//Moving status
	moveStatusLeftTopMotor:=LeftTopMotor.Status.Moving;
	moveStatusRightTopMotor:=RightTopMotor.Status.Moving;
	moveStatusLeftBottomMotor:=LeftBottomMotor.Status.Moving;
	moveStatusRightBottomMotor:=RightBottomMotor.Status.Moving;
	moveStatusAllAxisMotor:=moveStatusLeftTopMotor AND moveStatusRightTopMotor AND moveStatusLeftBottomMotor AND moveStatusRightBottomMotor;
	moveStatusAnyAxisMotor:=moveStatusLeftTopMotor OR moveStatusRightTopMotor OR moveStatusLeftBottomMotor OR moveStatusRightBottomMotor;
	//Velocity
	Velo_LeftTopMotor:=DINT_TO_LREAL(LREAL_TO_DINT(LeftTopMotor.NcToPlc.ActVelo*100000))/100000;
	Velo_RightTopMotor:=DINT_TO_LREAL(LREAL_TO_DINT(RightTopMotor.NcToPlc.ActVelo*100000))/100000;
	Velo_LeftBottomMotor:=DINT_TO_LREAL(LREAL_TO_DINT(LeftBottomMotor.NcToPlc.ActVelo*100000))/100000;
	Velo_RightBottomMotor:=DINT_TO_LREAL(LREAL_TO_DINT(RightBottomMotor.NcToPlc.ActVelo*100000))/100000;
	//LagDistance
	PosDiff_LeftTopMotor_actual:=DINT_TO_LREAL(LREAL_TO_DINT(LeftTopMotor.NcToPlc.PosDiff*100000))/100000;
	PosDiff_RightTopMotor_actual:=DINT_TO_LREAL(LREAL_TO_DINT(RightTopMotor.NcToPlc.PosDiff*100000))/100000;
	PosDiff_LeftBottomMotor_actual:=DINT_TO_LREAL(LREAL_TO_DINT(LeftBottomMotor.NcToPlc.PosDiff*100000))/100000;
	PosDiff_RightBottomMotor_actual:=DINT_TO_LREAL(LREAL_TO_DINT(RightBottomMotor.NcToPlc.PosDiff*100000))/100000;
	//Torque
	Torque_LeftTopMotor:=DINT_TO_LREAL(LREAL_TO_DINT(LeftTopMotor.NcToPlc.ActTorque*100000))/100000;
	Torque_RightTopMotor:=DINT_TO_LREAL(LREAL_TO_DINT(RightTopMotor.NcToPlc.ActTorque*100000))/100000;
	Torque_LeftBottomMotor:=DINT_TO_LREAL(LREAL_TO_DINT(LeftBottomMotor.NcToPlc.ActTorque*100000))/100000;
	Torque_RightBottomMotor:=DINT_TO_LREAL(LREAL_TO_DINT(RightBottomMotor.NcToPlc.ActTorque*100000))/100000;

	LeftTopMotor.ReadStatus();
	RightTopMotor.ReadStatus();
	LeftBottomMotor.ReadStatus();
	RightBottomMotor.ReadStatus();
	//
	//get Delta
	//
	//Delta Pos
	DeltaPos_LeftTop:=DINT_TO_LREAL(LREAL_TO_DINT((Pos_LeftTopLin - Pos_LeftTopMotor)*100000))/100000;
	DeltaPos_RightTop:=DINT_TO_LREAL(LREAL_TO_DINT((Pos_RightTopLin - Pos_RightTopMotor)*100000))/100000;
	DeltaPos_LeftBottom:=DINT_TO_LREAL(LREAL_TO_DINT((Pos_LeftBottomLin - Pos_LeftBottomMotor)*100000))/100000;
	DeltaPos_RightBottom:=DINT_TO_LREAL(LREAL_TO_DINT((Pos_RightBottomLin - Pos_RightBottomMotor)*100000))/100000;
	//Delta Velocity	
	DeltaVelo_LeftTop:=DINT_TO_LREAL(LREAL_TO_DINT((Velo_LeftTopLin - Velo_LeftTopMotor)*100000))/100000;
	DeltaVelo_RightTop:=DINT_TO_LREAL(LREAL_TO_DINT((Velo_RightTopLin - Velo_RightTopMotor)*100000))/100000;
	DeltaVelo_LeftBottom:=DINT_TO_LREAL(LREAL_TO_DINT((Velo_LeftBottomLin - Velo_LeftBottomMotor)*100000))/100000;
	DeltaVelo_RightBottom:=DINT_TO_LREAL(LREAL_TO_DINT((Velo_RightBottomLin - Velo_RightBottomMotor)*100000))/100000;
	//Delta lagDistance
	DeltaPosDiff_LeftTop_actual:=DINT_TO_LREAL(LREAL_TO_DINT((PosDiff_LeftTopLin_actual - PosDiff_LeftTopMotor_actual)*100000))/100000;
	DeltaPosDiff_RightTop_actual:=DINT_TO_LREAL(LREAL_TO_DINT((PosDiff_RightTopLin_actual - PosDiff_RightTopMotor_actual)*100000))/100000;
	DeltaPosDiff_LeftBottom_actual:=DINT_TO_LREAL(LREAL_TO_DINT((PosDiff_LeftBottomLin_actual - PosDiff_LeftBottomMotor_actual)*100000))/100000;
	DeltaPosDiff_RightBottom_actual:=DINT_TO_LREAL(LREAL_TO_DINT((PosDiff_RightBottomLin_actual - PosDiff_RightBottomMotor_actual)*100000))/100000;	
	//Delta Torque
	DeltaTorque_LeftTop:=DINT_TO_LREAL(LREAL_TO_DINT((Torque_LeftTopLin - Torque_LeftTopMotor)*100000))/100000;;
	DeltaTorque_RightTop:=DINT_TO_LREAL(LREAL_TO_DINT((Torque_RightTopLin - Torque_RightTopMotor)*100000))/100000;;
	DeltaTorque_LeftBottom:=DINT_TO_LREAL(LREAL_TO_DINT((Torque_LeftBottomLin -Torque_LeftBottomMotor)*100000))/100000;;
	DeltaTorque_RightBottom:=DINT_TO_LREAL(LREAL_TO_DINT((Torque_RightBottomLin - Torque_RightBottomMotor)*100000))/100000;;
	
	(*//feedback2 LE value when no LE*)
	IF NOT USELinearEncoder THEN
		Pos_LeftTop_2:=DINT_TO_LREAL(LREAL_TO_DINT((LeftTop_2.NcToPlc.ActPos+PositionBias_LeftTop)*100000))/100000;
		Pos_RightTop_2:=DINT_TO_LREAL(LREAL_TO_DINT((RightTop_2.NcToPlc.ActPos+PositionBias_RightTop)*100000))/100000;
		Pos_LeftBottom_2:=DINT_TO_LREAL(LREAL_TO_DINT((LeftBottom_2.NcToPlc.ActPos+PositionBias_LeftBottom)*100000))/100000;
		Pos_RightBottom_2:=DINT_TO_LREAL(LREAL_TO_DINT((RightBottom_2.NcToPlc.ActPos+PositionBias_RightBottom)*100000))/100000;
		Velo_LeftTop_2:=DINT_TO_LREAL(LREAL_TO_DINT(LeftTop_2.NcToPlc.ActVelo*100000))/100000;
		Velo_RightTop_2:=DINT_TO_LREAL(LREAL_TO_DINT(RightTop_2.NcToPlc.ActVelo*100000))/100000;
		Velo_LeftBottom_2:=DINT_TO_LREAL(LREAL_TO_DINT(LeftBottom_2.NcToPlc.ActVelo*100000))/100000;
		Velo_RightBottom_2:=DINT_TO_LREAL(LREAL_TO_DINT(RightBottom_2.NcToPlc.ActVelo*100000))/100000;
		LeftTop_2.ReadStatus();
		RightTop_2.ReadStatus();
		LeftBottom_2.ReadStatus();
		RightBottom_2.ReadStatus();
		PosDifference_LeftTop2to1:=Pos_LeftTop_2-Pos_LeftTopLin;
		PosDifference_RightTop2to1:=Pos_RightTop_2-Pos_RightTopLin;
		PosDifference_LeftBottom2to1:=Pos_LeftBottom_2-Pos_LeftBottomLin;
		PosDifference_RightBottom2to1:=Pos_RightBottom_2-Pos_RightBottomLin;
	END_IF
END_ACTION

ACTION A_InitRecipeParameters:
CASE state_loadParameters OF
	0:
		LoadParameter:=TRUE;
		Read_R_TRIG(CLK:=LoadParameter , Q=> );
		IF Read_R_TRIG.Q THEN
			state_loadParameters:=1;
		END_IF
	1:
		 ReturnDwordLoad:=RecipeManCommands.LoadAndWriteRecipe(RecipeDefinitionName:='Recipes' , RecipeName:='Parameters');
    	 LoadParameter:=FALSE;
		 IF ReturnDwordLoad<>0 THEN
		 	state_loadParameters:=-100;
		ELSE
			LoadRecipeParameters:=TRUE;
			LoadParameter:=FALSE;
			state_loadParameters:=88;
	 	END_IF
	88:
		loadParametersDone:=TRUE;
	-100:
		loadParametersDone:=FALSE;
		Error:=TRUE;
		ErrorId:=101;
		ErrorDescription:='LoadRecipeParameters Error';
		Plc_EmergencyStop:=FALSE;
END_CASE

//Save_R_TRIG(CLK:=SaveParameter , Q=> );
//IF Save_R_TRIG.Q THEN  //将plc数据以文件形式保存在工控机中
//	 RecipeManCommands.CreateRecipe(RecipeDefinitionName:='Recipes' , RecipeName:='Parameters' );
//	 RecipeManCommands.ReadAndSaveRecipe(RecipeDefinitionName:='Recipes' , RecipeName:='Parameters' );
//	 SaveParameter:=FALSE;
//END_IF
//Read_R_TRIG(CLK:=LoadParameter , Q=> );
//IF Read_R_TRIG.Q THEN  //将工控机中的文件数据读取到plc中
//     ReturnDwordLoad:=RecipeManCommands.LoadAndWriteRecipe(RecipeDefinitionName:='Recipes' , RecipeName:='Parameters');
//     LoadParameter:=FALSE;
//	 IF ReturnDwordLoad<>0 THEN
//		 Error:=TRUE;
//		 ErrorId:=101;
//		 ErrorDescription:='LoadRecipeParameters Error';
//		 Plc_EmergencyStop:=FALSE;
//	 END_IF
//END_IF
END_ACTION

ACTION A_KillOpcIocShellExe:
R_TRIG_Exekill(CLK:=bExe_Kill_Prog, Q=> );
CASE Exe_kill_step OF
	0:
		IF R_TRIG_Exekill.Q THEN
			NT_StartProcess_Kill.START:=FALSE;
			NT_StartProcess_Kill.PATHSTR:='C:\HZB\OpcIocShell\IDControlIOC\killcmd.bat';
			//NT_StartProcess_Kill.DIRNAME:='C:\Program Files (x86)\HZB\OpcIocShell\bin\opcIocShell.exe';
			Exe_kill_step:=10;
		END_IF;
	10:
		NT_StartProcess_Kill.START:=TRUE;
		Exe_kill_step:=20;
	20:
		IF NT_StartProcess_Kill.ERR THEN
			Exe_kill_step:=0;
		ELSE
			Exe_kill_step:=30;
		END_IF;

	30:
		NT_StartProcess_Kill.START:=TRUE;
		Exe_kill_step:=40;
	40:
		IF NOT NT_StartProcess_Kill.BUSY THEN
			NT_StartProcess_Kill.START:=FALSE;
			Exe_Kill_Done:=TRUE;
			Exe_kill_step:=0;
		END_IF;
END_CASE;

NT_StartProcess_Kill(
	NETID:='' ,
	PATHSTR:= ,
	DIRNAME:= , 
	COMNDLINE:= , 
	START:= ,
	ERRID=> );
END_ACTION

ACTION A_LED:
IF moveStatusAnyAxis THEN
	led_Run:=TRUE;
ELSE
	led_Run:=FALSE;
END_IF
IF Error THEN
	led_Error:=TRUE;
ELSE
	led_Error:=FALSE;
END_IF
END_ACTION

ACTION A_LEHeartBeatMonitor:
//monitor only while power on and not simulation or not use LE
IF NOT st_Power THEN
	RETURN;
END_IF
(**)
IF simulation THEN
	RETURN;
END_IF
IF NOT USELinearEncoder THEN
	RETURN;
END_IF

// 初始化
IF LEHeartBeatFirstScan THEN
    Velo_LeftTopLin_Last := LeftTopLin.NcToPlc.ActVelo;
    Velo_RightTopLin_Last := RightTopLin.NcToPlc.ActVelo;
    Velo_LeftBottomLin_Last := LeftBottomLin.NcToPlc.ActVelo;
    Velo_RightBottomLin_Last := RightBottomLin.NcToPlc.ActVelo;
    LEHeartBeatFirstScan := FALSE;
END_IF;

// 计算光栅前后速度差，速度差比位置差更敏感
DeltaVelo_LeftTopLin := ABS(LeftTopLin.NcToPlc.ActVelo - Velo_LeftTopLin_Last);
DeltaVelo_RightTopLin := ABS(RightTopLin.NcToPlc.ActVelo - Velo_RightTopLin_Last);
DeltaVelo_LeftBottomLin := ABS(LeftBottomLin.NcToPlc.ActVelo - Velo_LeftBottomLin_Last);
DeltaVelo_RightBottomLin := ABS(RightBottomLin.NcToPlc.ActVelo - Velo_RightBottomLin_Last);
//LeftTop monitor
IF DeltaVelo_LeftTopLin > LEHeartBeatDeadZone THEN
    // 有变动，光栅正常，计数器归零，更新位置,重置所有状态
    StableTimer_LeftTopLin(IN := FALSE, PT := LEHeartBeatAlarmTime);
    Alarm_LeftTopLin := FALSE;
    Velo_LeftTopLin_Last := LeftTopLin.NcToPlc.ActVelo;  // 
    StableTime_LeftTopLin := T#0S;
	IsInitialPositionSet_LeftTop:=FALSE;
	Alarm_LeftTopMotorPos:=FALSE;
	Alarm_LeftTopMotorVelo:=FALSE;
ELSE
    //一点变动没有了，光栅异常，开始计时
    StableTimer_LeftTopLin(
        IN := TRUE,
        PT := LEHeartBeatAlarmTime,
        ET => StableTime_LeftTopLin
    );
	//记录电机初始位置，后后续对比做准备
	IF NOT IsInitialPositionSet_LeftTop THEN
        Pos_LeftTopMotor_Initial := Pos_LeftTopMotor;  // 记录初始位置
        IsInitialPositionSet_LeftTop := TRUE;
   	END_IF;
    
    // 100ms速度完全不变，开始监控电机速度和位置
    IF StableTimer_LeftTopLin.Q THEN
        Alarm_LeftTopLin := TRUE;  // 
			//电机位置对比及监测
			MotorPosChange_LeftTop:=ABS( Pos_LeftTopMotor-Pos_LeftTopMotor_Initial);
			IF MotorPosChange_LeftTop > Threshold_LeftTopMotorPos THEN
				Alarm_LeftTopMotorPos:=TRUE;
				ErrorID:=5001;
				ErrorDescription:='5001';
				Error:=TRUE;
				FB_PlcEmergencyStop();
				LED_Error:=TRUE;
			ELSE
				Alarm_LeftTopMotorPos:=FALSE;
			END_IF
			//电机速度监测
			IF Velo_LeftTopMotor > Threshold_LeftTopMotorVelo THEN
				Alarm_LeftTopMotorVelo:=TRUE;
				ErrorID:=5002;
				ErrorDescription:='5002';
				Error:=TRUE;
				FB_PlcEmergencyStop();
				LED_Error:=TRUE;
			ELSE
				Alarm_LeftTopMotorVelo:=FALSE;
			END_IF
    ELSE
        Alarm_LeftTopLin := FALSE;
	END_IF
END_IF
//RightTop monitor
IF DeltaVelo_RightTopLin > LEHeartBeatDeadZone THEN
    // 有变动，光栅正常，计数器归零，更新位置,重置所有状态
    StableTimer_RightTopLin(IN := FALSE, PT := LEHeartBeatAlarmTime);
    Alarm_RightTopLin := FALSE;
    Velo_RightTopLin_Last := RightTopLin.NcToPlc.ActVelo;  // 
    StableTime_RightTopLin := T#0S;
	IsInitialPositionSet_RightTop:=FALSE;
	Alarm_RightTopMotorPos:=FALSE;
	Alarm_RightTopMotorVelo:=FALSE;
ELSE
    //一点变动没有了，光栅异常，开始计时
    StableTimer_RightTopLin(
        IN := TRUE,
        PT :=LEHeartBeatAlarmTime,
        ET => StableTime_RightTopLin
    );
	//记录电机初始位置，后后续对比做准备
	IF NOT IsInitialPositionSet_RightTop THEN
        Pos_RightTopMotor_Initial := Pos_RightTopMotor;  // 记录初始位置
        IsInitialPositionSet_RightTop := TRUE;
   	END_IF;
    
    // 100ms速度完全不变，开始监控电机速度和位置
    IF StableTimer_RightTopLin.Q THEN
        Alarm_RightTopLin := TRUE;  // 
			//电机位置对比及监测
			MotorPosChange_RightTop:=ABS( Pos_RightTopMotor-Pos_RightTopMotor_Initial);
			IF MotorPosChange_RightTop > Threshold_RightTopMotorPos THEN
				Alarm_RightTopMotorPos:=TRUE;
				ErrorID:=5003;
				ErrorDescription:='5003';
				Error:=TRUE;
				FB_PlcEmergencyStop();
				LED_Error:=TRUE;
			ELSE
				Alarm_RightTopMotorPos:=FALSE;
			END_IF
			//电机速度监测
			IF Velo_RightTopMotor > Threshold_RightTopMotorVelo THEN
				Alarm_RightTopMotorVelo:=TRUE;
				ErrorID:=5004;
				ErrorDescription:='5004';
				Error:=TRUE;
				FB_PlcEmergencyStop();
				LED_Error:=TRUE;
			ELSE
				Alarm_RightTopMotorVelo:=FALSE;
			END_IF
    ELSE
        Alarm_RightTopLin := FALSE;
	END_IF
END_IF
//LeftBottom monitor
IF DeltaVelo_LeftBottomLin > LEHeartBeatDeadZone THEN
    // 有变动，光栅正常，计数器归零，更新位置,重置所有状态
    StableTimer_LeftBottomLin(IN := FALSE, PT := LEHeartBeatAlarmTime);
    Alarm_LeftBottomLin := FALSE;
    Velo_LeftBottomLin_Last := LeftBottomLin.NcToPlc.ActVelo;  // 
    StableTime_LeftBottomLin := T#0S;
	IsInitialPositionSet_LeftBottom:=FALSE;
	Alarm_LeftBottomMotorPos:=FALSE;
	Alarm_LeftBottomMotorVelo:=FALSE;
ELSE
    //一点变动没有了，光栅异常，开始计时
    StableTimer_LeftBottomLin(
        IN := TRUE,
        PT := LEHeartBeatAlarmTime,
        ET => StableTime_LeftBottomLin
    );
	//记录电机初始位置，后后续对比做准备
	IF NOT IsInitialPositionSet_LeftBottom THEN
        Pos_LeftBottomMotor_Initial := Pos_LeftBottomMotor;  // 记录初始位置
        IsInitialPositionSet_LeftBottom := TRUE;
   	END_IF;
    
    // 100ms速度完全不变，开始监控电机速度和位置
    IF StableTimer_LeftBottomLin.Q THEN
        Alarm_LeftBottomLin := TRUE;  // 
			//电机位置对比及监测
			MotorPosChange_LeftBottom:=ABS( Pos_LeftBottomMotor-Pos_LeftBottomMotor_Initial);
			IF MotorPosChange_LeftBottom > Threshold_LeftBottomMotorPos THEN
				Alarm_LeftBottomMotorPos:=TRUE;
				ErrorID:=5005;
				ErrorDescription:='5005';
				Error:=TRUE;
				FB_PlcEmergencyStop();
				LED_Error:=TRUE;
			ELSE
				Alarm_LeftBottomMotorPos:=FALSE;
			END_IF
			//电机速度监测
			IF Velo_LeftBottomMotor > Threshold_LeftBottomMotorVelo THEN
				Alarm_LeftBottomMotorVelo:=TRUE;
				ErrorID:=5006;
				ErrorDescription:='5006';
				Error:=TRUE;
				FB_PlcEmergencyStop();
				LED_Error:=TRUE;
			ELSE
				Alarm_LeftBottomMotorVelo:=FALSE;
			END_IF
    ELSE
        Alarm_LeftBottomLin := FALSE;
	END_IF
END_IF
//RightBottom monitor
IF DeltaVelo_RightBottomLin > LEHeartBeatDeadZone THEN
    // 有变动，光栅正常，计数器归零，更新位置,重置所有状态
    StableTimer_RightBottomLin(IN := FALSE, PT := LEHeartBeatAlarmTime);
    Alarm_RightBottomLin := FALSE;
    Velo_RightBottomLin_Last := RightBottomLin.NcToPlc.ActVelo;  // 
    StableTime_RightBottomLin := T#0S;
	IsInitialPositionSet_RightBottom:=FALSE;
	Alarm_RightBottomMotorPos:=FALSE;
	Alarm_RightBottomMotorVelo:=FALSE;
ELSE
    //一点变动没有了，光栅异常，开始计时
    StableTimer_RightBottomLin(
        IN := TRUE,
        PT := LEHeartBeatAlarmTime,
        ET => StableTime_RightBottomLin
    );
	//记录电机初始位置，后后续对比做准备
	IF NOT IsInitialPositionSet_RightBottom THEN
        Pos_RightBottomMotor_Initial := Pos_RightBottomMotor;  // 记录初始位置
        IsInitialPositionSet_RightBottom := TRUE;
   	END_IF;
    
    // 100ms速度完全不变，开始监控电机速度和位置
    IF StableTimer_RightBottomLin.Q THEN
        Alarm_RightBottomLin := TRUE;  // 
			//电机位置对比及监测
			MotorPosChange_RightBottom:=ABS( Pos_RightBottomMotor-Pos_RightBottomMotor_Initial);
			IF MotorPosChange_RightBottom > Threshold_RightBottomMotorPos THEN
				Alarm_RightBottomMotorPos:=TRUE;
				ErrorID:=5007;
				ErrorDescription:='5007';
				Error:=TRUE;
				FB_PlcEmergencyStop();
				LED_Error:=TRUE;
			ELSE
				Alarm_RightBottomMotorPos:=FALSE;
			END_IF
			//电机速度监测
			IF Velo_RightBottomMotor > Threshold_RightBottomMotorVelo THEN
				Alarm_RightBottomMotorVelo:=TRUE;
				ErrorID:=5008;
				ErrorDescription:='5008';
				Error:=TRUE;
				FB_PlcEmergencyStop();
				LED_Error:=TRUE;
			ELSE
				Alarm_RightBottomMotorVelo:=FALSE;
			END_IF
    ELSE
        Alarm_RightBottomLin := FALSE;
	END_IF
END_IF
END_ACTION

ACTION A_LoadOpcIocShellExe:
R_TRIG_Exeload(CLK:=bExe_load_Prog, Q=> );
LoadOpcIocTON(PT:=T#10S);
CASE Exe_load_step OF
	0:
		LoadOpcIocTON.IN:=TRUE;
		IF R_TRIG_Exeload.Q THEN
			NT_StartProcess_Load.START:=FALSE;
			NT_StartProcess_Load.PATHSTR:='C:\HZB\OpcIocShell\IDControlIOC\startTwinCATOPCServer.bat';
			Exe_load_step:=10;
		END_IF;
	10:
		IF LoadOpcIocTON.Q THEN
			NT_StartProcess_Load.START:=TRUE;
			Exe_load_step:=20;
		END_IF
	20:
		LoadOpcIocTON.IN:=FALSE;
		IF NT_StartProcess_Load.ERR THEN
			Exe_load_step:=0;
		ELSE
			Exe_load_step:=30;
		END_IF;
	30:
		IF NOT NT_StartProcess_Load.BUSY THEN
			NT_StartProcess_Load.START:=FALSE;
			Exe_Load_Done:=TRUE;
			Exe_load_step:=0;
		END_IF;
END_CASE;

NT_StartProcess_Load(
	NETID:='' ,
	PATHSTR:= ,
	DIRNAME:= , 
	COMNDLINE:= , 
	START:= ,
	ERRID=> );
END_ACTION

ACTION A_MonitorMotorAndLE:
//Monitoring Motor and LE Position/Velocity
IF 	ABS(DeltaPos_LeftTop) > ThresholdDeltaPos_LeftTop THEN
	ErrorID:=6001;
	Error:=TRUE;
	ErrorDescription:='ABS(DeltaPos_LeftTop) > ThresholdDeltaPos_LeftTop';
	FB_PlcEmergencyStop();
	LED_Error:=TRUE;
END_IF
IF ABS(DeltaPos_RightTop) > ThresholdDeltaPos_RightTop THEN
	ErrorID:=6002;
	Error:=TRUE;
	ErrorDescription:='ABS(DeltaPos_RightTop) > ThresholdDeltaPos_RightTop';
	FB_PlcEmergencyStop();
	LED_Error:=TRUE;
END_IF
IF ABS(DeltaPos_LeftBottom) > ThresholdDeltaPos_LeftBottom THEN
	ErrorID:=6003;
	Error:=TRUE;
	ErrorDescription:='ABS(DeltaPos_LeftBottom) > ThresholdDeltaPos_LeftBottom';
	FB_PlcEmergencyStop();
	LED_Error:=TRUE;
END_IF
IF ABS(DeltaPos_RightBottom) > ThresholdDeltaPos_RightBottom THEN
	ErrorID:=6004;
	Error:=TRUE;
	ErrorDescription:='ABS(DeltaPos_RightBottom) > ThresholdDeltaPos_RightBottom';
	FB_PlcEmergencyStop();
	LED_Error:=TRUE;
END_IF

IF ABS(DeltaVelo_LeftTop) > ThresholdDeltaVelo_LeftTop THEN
	ErrorID:=6005;
	Error:=TRUE;
	ErrorDescription:='ABS(DeltaVelo_LeftTop) > ThresholdDeltaVelo_LeftTop';
	FB_PlcEmergencyStop();
	LED_Error:=TRUE;
END_IF
IF ABS(DeltaVelo_RightTop) > ThresholdDeltaVelo_RightTop THEN
	ErrorID:=6006;
	Error:=TRUE;
	ErrorDescription:='ABS(DeltaVelo_RightTop) > ThresholdDeltaVelo_RightTop';
	FB_PlcEmergencyStop();
	LED_Error:=TRUE;
END_IF
IF ABS(DeltaVelo_LeftBottom) > ThresholdDeltaVelo_LeftBottom THEN
	ErrorID:=6007;
	Error:=TRUE;
	ErrorDescription:='ABS(DeltaVelo_LeftBottom) > ThresholdDeltaVelo_LeftBottom';
	FB_PlcEmergencyStop();
	LED_Error:=TRUE;
END_IF
IF ABS(DeltaVelo_RightBottom) > ThresholdDeltaVelo_RightBottom THEN
	ErrorID:=6008;
	Error:=TRUE;
	ErrorDescription:='ABS(DeltaVelo_RightBottom) > ThresholdDeltaVelo_RightBottom';
	FB_PlcEmergencyStop();
	LED_Error:=TRUE;
END_IF

(*
//
//IF NotMoving ,Threshold is less
//
IF NOT moveStatusLeftTop THEN
		IF 	ABS(DeltaPos_LeftTop) > ThresholdDeltaPos_LeftTop/3 THEN
		ErrorID:=6009;
		Error:=TRUE;
		ErrorDescription:='ABS(DeltaPos_LeftTop) > ThresholdDeltaPos_LeftTop/3';
		FB_PlcEmergencyStop();
		LED_Error:=TRUE;
	END_IF
END_IF
IF NOT moveStatusRightTop THEN
	IF ABS(DeltaPos_RightTop) > ThresholdDeltaPos_RightTop/3 THEN
		ErrorID:=6010;
		Error:=TRUE;
		ErrorDescription:='ABS(DeltaPos_RightTop) > ThresholdDeltaPos_RightTop/3';
		FB_PlcEmergencyStop();
		LED_Error:=TRUE;
	END_IF
END_IF
IF NOT moveStatusLeftBottom THEN
	IF ABS(DeltaPos_LeftBottom) > ThresholdDeltaPos_LeftBottom/3 THEN
		ErrorID:=6011;
		Error:=TRUE;
		ErrorDescription:='ABS(DeltaPos_LeftBottom) > ThresholdDeltaPos_LeftBottom/3';
		FB_PlcEmergencyStop();
		LED_Error:=TRUE;
	END_IF
END_IF
IF NOT moveStatusRightBottom THEN
	IF ABS(DeltaPos_RightBottom) > ThresholdDeltaPos_RightBottom/3 THEN
		ErrorID:=6012;
		Error:=TRUE;
		ErrorDescription:='ABS(DeltaPos_RightBottom) > ThresholdDeltaPos_RightBottom';
		FB_PlcEmergencyStop();
		LED_Error:=TRUE;
	END_IF
END_IF

//
IF NOT moveStatusLeftTop THEN
	IF ABS(DeltaVelo_LeftTop) > ThresholdDeltaVelo_LeftTop/3 THEN
		ErrorID:=6013;
		Error:=TRUE;
		ErrorDescription:='ABS(DeltaVelo_LeftTop) > ThresholdDeltaVelo_LeftTop/3';
		FB_PlcEmergencyStop();
		LED_Error:=TRUE;
	END_IF
END_IF
IF NOT moveStatusRightTop THEN
	IF ABS(DeltaVelo_RightTop) > ThresholdDeltaVelo_RightTop/3 THEN
		ErrorID:=6014;
		Error:=TRUE;
		ErrorDescription:='ABS(DeltaVelo_RightTop) > ThresholdDeltaVelo_RightTop/3';
		FB_PlcEmergencyStop();
		LED_Error:=TRUE;
	END_IF
END_IF
IF NOT moveStatusLeftBottom THEN
	IF ABS(DeltaVelo_LeftBottom) > ThresholdDeltaVelo_LeftBottom/3 THEN
		ErrorID:=6015;
		Error:=TRUE;
		ErrorDescription:='ABS(DeltaVelo_LeftBottom) > ThresholdDeltaVelo_LeftBottom/3';
		FB_PlcEmergencyStop();
		LED_Error:=TRUE;
	END_IF
END_IF
IF NOT moveStatusRightBottom THEN
	IF ABS(DeltaVelo_RightBottom) > ThresholdDeltaVelo_RightBottom/3 THEN
		ErrorID:=6016;
		Error:=TRUE;
		ErrorDescription:='ABS(DeltaVelo_RightBottom) > ThresholdDeltaVelo_RightBottom/3';
		FB_PlcEmergencyStop();
		LED_Error:=TRUE;
	END_IF
END_IF
*)
END_ACTION

ACTION A_PosDiffDetectiion:
IF ABS(PosDiff_LeftTopLin_actual)>PosDiff_LeftTopLin THEN
	ErrorID:=201;
	Error:=TRUE;
	ErrorDescription:='ABS(PosDiff_LeftTopLin_actual)>PosDiff_LeftTopLin';
	FB_PlcEmergencyStop();
	LED_Error:=TRUE;
END_IF
IF ABS(PosDiff_RightTopLin_actual)>PosDiff_RightTopLin THEN
	ErrorID:=202;
	Error:=TRUE;
	ErrorDescription:='ABS(PosDiff_RightTopLin_actual)>PosDiff_RightTopLin';
	FB_PlcEmergencyStop();
	LED_Error:=TRUE;
END_IF
IF ABS(PosDiff_LeftBottomLin_actual)>PosDiff_LeftBottomLin THEN
	ErrorID:=203;
	Error:=TRUE;
	ErrorDescription:='ABS(PosDiff_LeftBottomLin_actual)>PosDiff_LeftBottomLin';
	FB_PlcEmergencyStop();
	LED_Error:=TRUE;
END_IF
IF ABS(PosDiff_RightBottomLin_actual)>PosDiff_RightBottomLin THEN
	ErrorID:=204;
	ErrorDescription:='ABS(PosDiff_RightBottomLin_actual)>PosDiff_RightBottomLin';
	Error:=TRUE;
	FB_PlcEmergencyStop();
	LED_Error:=TRUE;
END_IF
//
IF ABS(PosDiff_LeftTopLin_actual-PosDiff_RightTopLin_actual)>0.05 THEN
	ErrorID:=205;
	ErrorDescription:='ABS(PosDiff_LeftTopLin_actual-PosDiff_RightTopLin_actual)>0.05';
	Error:=TRUE;
	FB_PlcEmergencyStop();
	LED_Error:=TRUE;
ELSIF ABS(PosDiff_LeftBottomLin_actual-PosDiff_RightBottomLin_actual)>0.05 THEN
	ErrorID:=206;
	ErrorDescription:='ABS(PosDiff_LeftBottomLin_actual-PosDiff_RightBottomLin_actual)>0.05';
	Error:=TRUE;
	FB_PlcEmergencyStop();
	LED_Error:=TRUE;
END_IF
END_ACTION

ACTION A_RestartDrivers:
Relay_EL2624[0]:=btn_RestartDriver1;
Relay_EL2624[1]:=btn_RestartDriver2;
Relay_EL2624[2]:=btn_RestartDriver3;
Relay_EL2624[3]:=btn_RestartDriver4;
Relay_EL2624[4]:=btn_RestartDriver5;
Relay_EL2624[5]:=btn_RestartDriver6;
Relay_EL2624[6]:=btn_RestartDriver7;
Relay_EL2624[7]:=btn_RestartDriver8;
///
//1.上升沿触发，btn_RestartDrivers上升沿后，btn_RestartDriver1~8全部高电平
//2、3s后，Driver1~8全部恢复低电平
//3、恢复全部状态到初始
///
RestartDriver_RTRIG(CLK:=btn_RestartDriversAll);
IF RestartDriver_RTRIG.Q THEN
	RestartDriver_Triggered:=TRUE;
	RestartDriver_Done:=FALSE;
END_IF
IF RestartDriver_Triggered THEN
	CASE RestartDriver_State OF
		0:
			btn_RestartDriver1:=TRUE;
			btn_RestartDriver2:=TRUE;
			btn_RestartDriver3:=TRUE;
			btn_RestartDriver4:=TRUE;
			btn_RestartDriver5:=TRUE;
			btn_RestartDriver6:=TRUE;
			btn_RestartDriver7:=TRUE;
			btn_RestartDriver8:=TRUE;
			//计时开始
			RestartDriver_TON(PT:=T#10S);
			RestartDriver_TON.IN:=TRUE;
			IF RestartDriver_TON.Q THEN
				RestartDriver_State:=1;
			END_IF
		1:
			btn_RestartDriver1:=FALSE;
			btn_RestartDriver2:=FALSE;
			btn_RestartDriver3:=FALSE;
			btn_RestartDriver4:=FALSE;
			btn_RestartDriver5:=FALSE;
			btn_RestartDriver6:=FALSE;
			btn_RestartDriver7:=FALSE;
			btn_RestartDriver8:=FALSE;
			RestartDriver_State:=88;
		88:
			RestartDriver_TON.IN:=FALSE;
			btn_RestartDriversAll:=FALSE;
			RestartDriver_State:=0;
			RestartDriver_Triggered:=FALSE;
			RestartDriver_Done:=TRUE;
	END_CASE
END_IF
END_ACTION

ACTION A_RestartTC:
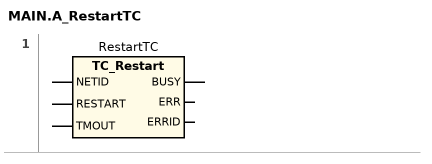
// NETWORK 1
RestartTC(); // TC_Restart
END_ACTION

ACTION A_SafePlcStartInit:
fb_ton0(PT:=t#1s);
fb_ton1(PT:=t#0.1s);
fb_ton2(PT:=t#0.1s);
fb_ton3(PT:=t#0.1s);

CASE SafeStatus OF
	0:
		IF COM_ERROR OR NOT Estop_Out THEN
			Err_Ack:=TRUE;
			fb_ton0.IN:=TRUE;
			SafeStatus:=1;
		ELSE
			SafePLCRunOK:=TRUE;
			SafeStatus:=0;
		END_IF
	1:
		IF fb_ton0.Q THEN
			Err_Ack:=FALSE;
			Safe_run:=TRUE;
			fb_ton1.IN:=TRUE;
			SafeStatus:=2;
		END_IF

	2:
		IF fb_ton1.Q THEN
			IF Estop_RunAndRestart=FALSE THEN
				Estop_RunAndRestart:=TRUE;
				fb_ton2.IN:=TRUE;
				SafeStatus:=3;
			END_IF
		END_IF
	3:
		IF fb_ton2.Q THEN
			IF Estop_RunAndRestart THEN
				Estop_RunAndRestart:=FALSE;
				fb_ton3.IN:=TRUE;
				SafeStatus:=4;
			END_IF
		END_IF
	4:
		IF fb_ton3.Q THEN
			IF Estop_Out THEN
				SafePLCRunOK:=TRUE;
				SafeStatus:=0;
			ELSE
				SafePLCRunOK:=FALSE;
				//Error:=TRUE;
				//ErrorId:=301;
				//ErrorDescription:='SafePLCRunOK fail';
			END_IF
		fb_ton0.IN:=FALSE;
		fb_ton1.IN:=FALSE;
		fb_ton2.IN:=FALSE;
		fb_ton3.IN:=FALSE;
		END_IF


END_CASE
END_ACTION

ACTION A_SetAxisPosition:
fb_ton4(PT:=t#0.5s);
CASE SetAxisPosState OF
	0:	(*FB_Set_AxisPosition*)
		FB_Set_AxisPosition(Execute:=TRUE);
		fb_ton4.IN:=TRUE;
		SetAxisPosState:=1;
	1:	(*wait*)
		FB_Set_AxisPosition();
		IF NOT FB_Set_AxisPosition.Done THEN		
			IF NOT fb_ton4.Q THEN
				SetAxisPosState:=1;
			ELSE
				SetAxisPosState:=99;
			END_IF
		ELSE
			SetAxisPosState:=88;
		END_IF
	88:
		SetAxisPosState:=0;
		SerAxisPositionDone:=TRUE;
		Error:=FALSE;
		ErrorID:=0;
		FB_Set_AxisPosition.Execute:=FALSE;
		fb_ton4.IN:=FALSE;
	99:
		SetAxisPosState:=99;
		SerAxisPositionDone:=FALSE;
		Error:=TRUE;
		FB_Set_AxisPosition.Execute:=FALSE;
		fb_ton4.IN:=FALSE;
		LED_Error:=TRUE;
		ErrorID:=401;
		ErrorDescription:='SetAxisPosition fail';
END_CASE
END_ACTION

ACTION A_SetLinearEncoderPositionBias:
//No LE
IF NOT USELinearEncoder THEN
	PositionBias_LeftTopLin:=0;
	PositionBias_RightTopLin:=0;
	PositionBias_LeftBottomLin:=0;
	PositionBias_RightBottomLin:=0;
END_IF
//没有传感器OR不是CPMU不低温补偿OR低温不到位，均不补偿
IF HasTemperatureSensorOrNot AND CryogenicCompensationOn THEN
	PositionBias_LeftTopLin:=PositionBias_LeftTop+CryogenicCompensation_LeftTop;
	PositionBias_RightTopLin:=PositionBias_RightTop+CryogenicCompensation_RightTop;
	PositionBias_LeftBottomLin:=PositionBias_LeftBottom+CryogenicCompensation_LeftBottom;
	PositionBias_RightBottomLin:=PositionBias_RightBottom+CryogenicCompensation_RightBottom;
	CryogenicCompensationDone:=TRUE;
ELSE
	PositionBias_LeftTopLin:=PositionBias_LeftTop;
	PositionBias_RightTopLin:=PositionBias_RightTop;
	PositionBias_LeftBottomLin:=PositionBias_LeftBottom;
	PositionBias_RightBottomLin:=PositionBias_RightBottom;
END_IF

//设置bias开始
A_SetLinearEncoderPositionBiasMC();
PositionBiasTON(PT:=T#0.1S);
CASE state_setLEPosBias OF
	0:
		PositionBiasTON.IN:=TRUE;
		IF MC_SetLEPosBias_LeftTop.Error OR MC_SetLEPosBias_RightTop.Error OR 
			MC_SetLEPosBias_LeftBottom.Error OR MC_SetLEPosBias_RightBottom.Error THEN
			state_setLEPosBias:=-100;
		ELSE 
			state_setLEPosBias:=1;
		END_IF
	1:
		IF NOT MC_SetLEPosBias_LeftTop.Done OR NOT MC_SetLEPosBias_RightTop.Done OR 
			NOT MC_SetLEPosBias_LeftBottom.Done OR NOT MC_SetLEPosBias_RightBottom.Done THEN
			MC_SetLEPosBias_LeftTop.Execute:=TRUE;
			MC_SetLEPosBias_RightTop.Execute:=TRUE;
			MC_SetLEPosBias_LeftBottom.Execute:=TRUE;
			MC_SetLEPosBias_RightBottom.Execute:=TRUE;
			state_setLEPosBias:=2;
		ELSE
			state_setLEPosBias:=-100;
		END_IF
	2:
		IF NOT MC_SetLEPosBias_LeftTop.Done OR NOT MC_SetLEPosBias_RightTop.Done OR 
			NOT MC_SetLEPosBias_LeftBottom.Done OR NOT MC_SetLEPosBias_RightBottom.Done THEN
			IF NOT PositionBiasTON.Q THEN
				state_setLEPosBias:=2;
			ELSE
				state_setLEPosBias:=-100;
			END_IF
		END_IF
		IF  MC_SetLEPosBias_LeftTop.Done AND MC_SetLEPosBias_RightTop.Done AND
			MC_SetLEPosBias_LeftBottom.Done AND MC_SetLEPosBias_RightBottom.Done THEN
			state_setLEPosBias:=88;
		END_IF	
		IF MC_SetLEPosBias_LeftTop.Error OR MC_SetLEPosBias_RightTop.Error OR 
			MC_SetLEPosBias_LeftBottom.Error OR MC_SetLEPosBias_RightBottom.Error THEN
			state_setLEPosBias:=-100;
		END_IF 
		
	88:
		PositionBiasTON.IN:=FALSE;
		PositionBiasDone:=TRUE;
	-100:
		PositionBiasTON.IN:=FALSE;
		PositionBiasDone:=FALSE;
		Error:=TRUE;
		ErrorId:=901;
		ErrorDescription:='Set LinearEncoderPositionBias Error';
		Plc_EmergencyStop:=FALSE;
END_CASE
END_ACTION

ACTION A_SetLinearEncoderPositionBiasMC:
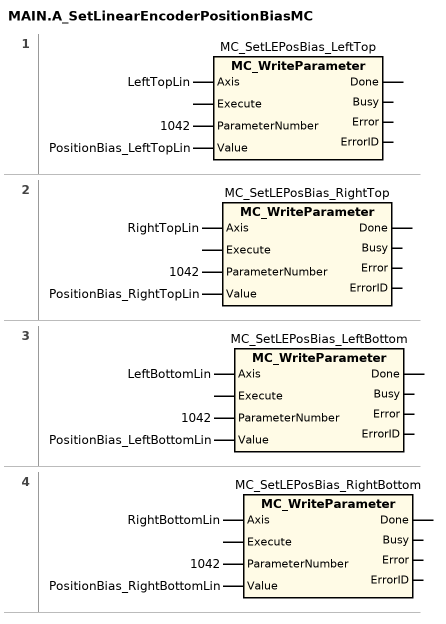
// NETWORK 1
MC_SetLEPosBias_LeftTop(Axis := LeftTopLin, ParameterNumber := 1042, Value := PositionBias_LeftTopLin); // MC_WriteParameter

// NETWORK 2
MC_SetLEPosBias_RightTop(Axis := RightTopLin, ParameterNumber := 1042, Value := PositionBias_RightTopLin); // MC_WriteParameter

// NETWORK 3
MC_SetLEPosBias_LeftBottom(
    Axis := LeftBottomLin,
    ParameterNumber := 1042,
    Value := PositionBias_LeftBottomLin); // MC_WriteParameter

// NETWORK 4
MC_SetLEPosBias_RightBottom(
    Axis := RightBottomLin,
    ParameterNumber := 1042,
    Value := PositionBias_RightBottomLin); // MC_WriteParameter
END_ACTION

ACTION A_SetMotorAxisPosition:
fb_ton4_2(PT:=T#0.5S);
CASE SetMotorAxisPosState OF
	0:	(*FB_Set_AxisPosition*)
		FB_Set_MotorAxisPosition(Execute:=TRUE);
		fb_ton4_2.IN:=TRUE;
		SetMotorAxisPosState:=1;
	1:	(*wait*)
		FB_Set_MotorAxisPosition();
		IF NOT FB_Set_MotorAxisPosition.Done THEN		
			IF NOT fb_ton4_2.Q THEN
				SetMotorAxisPosState:=1;
			ELSE
				SetMotorAxisPosState:=99;
			END_IF
		ELSE
			SetMotorAxisPosState:=88;
		END_IF
	88:
		SetMotorAxisPosState:=0;
		SetMotorAxisPositionDone:=TRUE;
		Error:=FALSE;
		ErrorID:=0;
		FB_Set_MotorAxisPosition.Execute:=FALSE;
		fb_ton4_2.IN:=FALSE;
	99:
		SetMotorAxisPosState:=99;
		SetMotorAxisPositionDone:=FALSE;
		Error:=TRUE;
		FB_Set_MotorAxisPosition.Execute:=FALSE;
		fb_ton4.IN:=FALSE;
		LED_Error:=TRUE;
		ErrorID:=401;
		ErrorDescription:='SetMotorAxisPosition fail';
END_CASE
END_ACTION

END_PROGRAM

// ---- POUs/CommonFB/MainFB/FB_SetAxisPosition.TcPOU
(****************************************************************
NAME:			FB_SetAxisPosition
DATA:			2017.2.16
VERSION:		1.0.0
DESCRIPTION:	FB_SetAxisPosition
HISTORY:
				2017.2.16		NEW

***************************************************************)
FUNCTION_BLOCK FB_SetAxisPosition
VAR_INPUT
	//GapValueSet:LREAL:=0;
	ValueSet_LeftTop:LREAL:=0;
	ValueSet_RightTop:LREAL:=0;
	ValueSet_LeftBottom:LREAL:=0;
	ValueSet_RightBottom:LREAL:=0;
	Execute:BOOL;
END_VAR
VAR_OUTPUT
	FbID:DINT:=1001;
	State:DINT;
	Busy:BOOL;
	Done:BOOL;
	Error:BOOL;
	ErrorID:DINT;
END_VAR
VAR
	LeftTopLin_MC_SetPosition: MC_SetPosition;
	RightTopLin_MC_SetPosition: MC_SetPosition;
	LeftBottomLin_MC_SetPosition: MC_SetPosition;
	RightBottomLin_MC_SetPosition: MC_SetPosition;
	fb_ton: TON;
	FB_Couple_Axis: FB_CoupleAxis;
	FB_PlcEmergencyStop: FB_PlcEmergencyStop;
END_VAR

IF Execute THEN
Busy:=TRUE;
Done:=FALSE;
fb_ton(PT:=t#0.1s);
CASE State OF
	0:
		IF LeftTopLin_MC_SetPosition.Error OR RightTopLin_MC_SetPosition.Error
			OR LeftBottomLin_MC_SetPosition.Error OR RightBottomLin_MC_SetPosition.Error THEN		(*FB Error*)
			ErrorID:=1;
			State:=99;
		ELSIF FB_Couple_Axis.InGear THEN		
			ErrorID:=2;
			State:=99;
		ELSIF LeftTopLin.NcToPlc.CoupleState=0 AND LeftBottomLin.NcToPlc.CoupleState=0
			AND RightTopLin.NcToPlc.CoupleState=0 AND RightBottomLin.NcToPlc.CoupleState=0 THEN	
			State:=1;
		ELSE
			ErrorID:=3;
			State:=-100;
		END_IF
	1:	(*Execute*)
		LeftTopLin_MC_SetPosition.Position:=ValueSet_LeftTop;
		LeftTopLin_MC_SetPosition.Execute:=TRUE;
		RightTopLin_MC_SetPosition.Position:=ValueSet_RightTop;
		RightTopLin_MC_SetPosition.Execute:=TRUE;
		LeftBottomLin_MC_SetPosition.Position:=ValueSet_LeftBottom;
		LeftBottomLin_MC_SetPosition.Execute:=TRUE;
		RightBottomLin_MC_SetPosition.Position:=ValueSet_RightBottom;
		RightBottomLin_MC_SetPosition.Execute:=TRUE;
		A_SetPositionMC();
		fb_ton.IN:=TRUE;
		State:=2;
	2:	(*Wait*)
		A_SetPositionMC();
		IF NOT LeftTopLin_MC_SetPosition.Done OR NOT RightTopLin_MC_SetPosition.Done
			OR NOT LeftBottomLin_MC_SetPosition.Done OR NOT RightBottomLin_MC_SetPosition.Done THEN		
			IF NOT fb_ton.Q THEN
				State:=2;
			ELSE
				ErrorID:=4;
				State:=99;
			END_IF
		ELSIF  LeftTopLin_MC_SetPosition.Done AND RightTopLin_MC_SetPosition.Done
			AND LeftBottomLin_MC_SetPosition.Done AND RightBottomLin_MC_SetPosition.Done THEN		
			State:=88;
		ELSE
			ErrorID:=5;
			State:=99;
		END_IF
	88:
		Execute:=FALSE;
		State:=0;
		Busy:=FALSE;
		Done:=TRUE;
		Error:=FALSE;
		ErrorID:=0;
		LeftTopLin_MC_SetPosition.Execute:=FALSE;
		RightTopLin_MC_SetPosition.Execute:=FALSE;
		LeftBottomLin_MC_SetPosition.Execute:=FALSE;
		RightBottomLin_MC_SetPosition.Execute:=FALSE;
		fb_ton.IN:=FALSE;
	99:
		Execute:=FALSE;
		State:=99;
		Busy:=FALSE;
		Done:=FALSE;
		Error:=TRUE;
		LeftTopLin_MC_SetPosition.Execute:=FALSE;
		RightTopLin_MC_SetPosition.Execute:=FALSE;
		LeftBottomLin_MC_SetPosition.Execute:=FALSE;
		RightBottomLin_MC_SetPosition.Execute:=FALSE;
		fb_ton.IN:=FALSE;
	-100:
		FB_PlcEmergencyStop();
		Execute:=FALSE;
		State:=-100;
		Busy:=FALSE;
		Done:=FALSE;
		Error:=TRUE;
		LeftTopLin_MC_SetPosition.Execute:=FALSE;
		RightTopLin_MC_SetPosition.Execute:=FALSE;
		LeftBottomLin_MC_SetPosition.Execute:=FALSE;
		RightBottomLin_MC_SetPosition.Execute:=FALSE;
		fb_ton.IN:=FALSE;
END_CASE
END_IF

ACTION A_SetPositionMC:
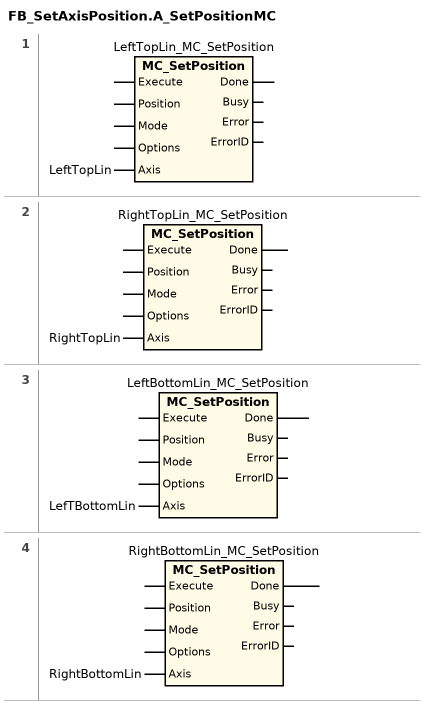
// NETWORK 1
LeftTopLin_MC_SetPosition(Axis := LeftTopLin); // MC_SetPosition

// NETWORK 2
RightTopLin_MC_SetPosition(Axis := RightTopLin); // MC_SetPosition

// NETWORK 3
LeftBottomLin_MC_SetPosition(Axis := LefTBottomLin); // MC_SetPosition

// NETWORK 4
RightBottomLin_MC_SetPosition(Axis := RightBottomLin); // MC_SetPosition
END_ACTION

END_FUNCTION_BLOCK

